ABB RAPID module: P50.mod

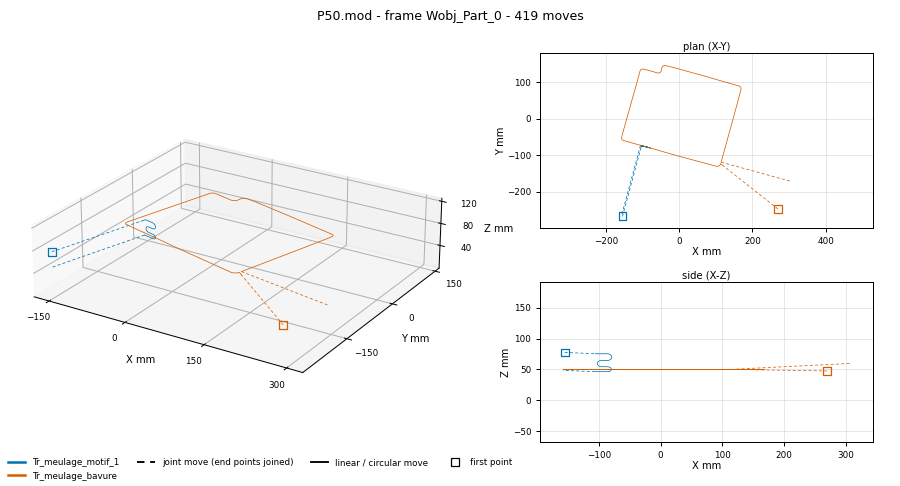
[picture p0: tool path of P50.mod in frame Wobj_Part_0, 419 of 426 moves have a stored position in this frame; points joined in program order, loops and branches not executed]
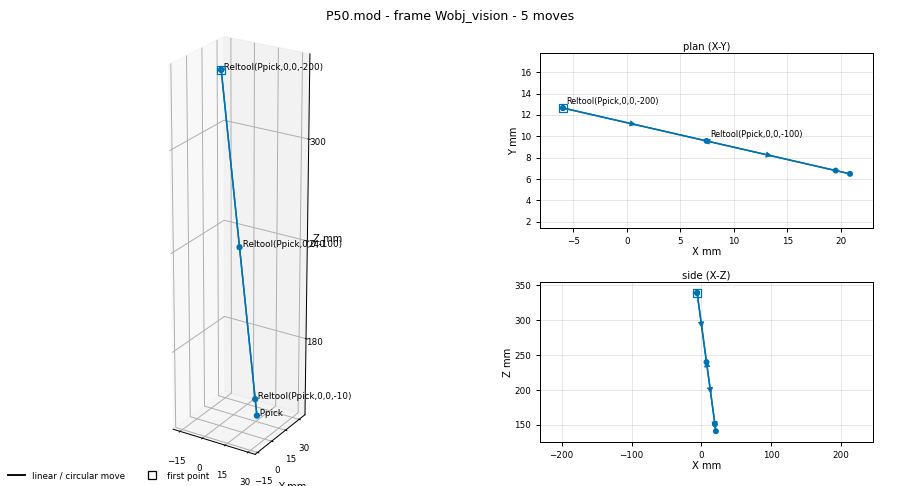
[picture p1: tool path of P50.mod in frame Wobj_vision, 5 of 426 moves have a stored position in this frame; points joined in program order, loops and branches not executed]
MODULE P50
	LOCAL CONST Speeddata vitesse_Tronconnage :=[10, 500, 0, 0];
	LOCAL CONST Robtarget Tr_meulage_motif_1_App1 :=[[-155.319755166464,-266.991909099729,77.372571942786],[0.697372246118371,-0.704623915003405,0.0931525017095072,-0.0921938185257175],[0,0,0,0],[8.999999E+09,8.999999E+09,8.999999E+09,8.999999E+09,8.999999E+09,8.999999E+09]];
	LOCAL CONST Robtarget Tr_meulage_motif_1_App2 :=[[-105.948658461448,-83.5290196737364,75.4071168783893],[0.697372246118371,-0.704623915003405,0.0931525017095072,-0.0921938185257175],[0,0,0,0],[8.999999E+09,8.999999E+09,8.999999E+09,8.999999E+09,8.999999E+09,8.999999E+09]];
	LOCAL CONST Robtarget Tr_meulage_motif_1_P0 :=[[-103.3501796875,-73.873078125,75.303671875],[0.697372246118371,-0.704623915003405,0.0931525017095072,-0.0921938185257175],[0,0,0,0],[8.999999E+09,8.999999E+09,8.999999E+09,8.999999E+09,8.999999E+09,8.999999E+09]];
	LOCAL CONST Robtarget Tr_meulage_motif_1_P1 :=[[-102.3816328125,-74.12190625,75.303671875],[0.697372246118371,-0.704623915003405,0.0931525017095072,-0.0921938185257175],[0,0,0,0],[8.999999E+09,8.999999E+09,8.999999E+09,8.999999E+09,8.999999E+09,8.999999E+09]];
	LOCAL CONST Robtarget Tr_meulage_motif_1_P2 :=[[-101.4130859375,-74.3707421875,75.303671875],[0.697372246118371,-0.704623915003405,0.0931525017095072,-0.0921938185257175],[0,0,0,0],[8.999999E+09,8.999999E+09,8.999999E+09,8.999999E+09,8.999999E+09,8.999999E+09]];
	LOCAL CONST Robtarget Tr_meulage_motif_1_P3 :=[[-100.4445390625,-74.6195703125,75.303671875],[0.697372246118371,-0.704623915003405,0.0931525017095072,-0.0921938185257175],[0,0,0,0],[8.999999E+09,8.999999E+09,8.999999E+09,8.999999E+09,8.999999E+09,8.999999E+09]];
	LOCAL CONST Robtarget Tr_meulage_motif_1_P4 :=[[-99.4759921875,-74.8683984375,75.303671875],[0.697372246118371,-0.704623915003405,0.0931525017095072,-0.0921938185257175],[0,0,0,0],[8.999999E+09,8.999999E+09,8.999999E+09,8.999999E+09,8.999999E+09,8.999999E+09]];
	LOCAL CONST Robtarget Tr_meulage_motif_1_P5 :=[[-98.5074453125,-75.117234375,75.303671875],[0.697372246118371,-0.704623915003405,0.0931525017095072,-0.0921938185257175],[0,0,0,0],[8.999999E+09,8.999999E+09,8.999999E+09,8.999999E+09,8.999999E+09,8.999999E+09]];
	LOCAL CONST Robtarget Tr_meulage_motif_1_P6 :=[[-97.5388984375,-75.3660625,75.303671875],[0.697372246118371,-0.704623915003405,0.0931525017095072,-0.0921938185257175],[0,0,0,0],[8.999999E+09,8.999999E+09,8.999999E+09,8.999999E+09,8.999999E+09,8.999999E+09]];
	LOCAL CONST Robtarget Tr_meulage_motif_1_P7 :=[[-96.5703515625,-75.6148984375,75.303671875],[0.697372246118371,-0.704623915003405,0.0931525017095072,-0.0921938185257175],[0,0,0,0],[8.999999E+09,8.999999E+09,8.999999E+09,8.999999E+09,8.999999E+09,8.999999E+09]];
	LOCAL CONST Robtarget Tr_meulage_motif_1_P8 :=[[-95.6018046875,-75.8637265625,75.303671875],[0.697372246118371,-0.704623915003405,0.0931525017095072,-0.0921938185257175],[0,0,0,0],[8.999999E+09,8.999999E+09,8.999999E+09,8.999999E+09,8.999999E+09,8.999999E+09]];
	LOCAL CONST Robtarget Tr_meulage_motif_1_P9 :=[[-94.6332578125,-76.1125546875,75.3036796875],[0.697372246118371,-0.704623915003405,0.0931525017095072,-0.0921938185257175],[0,0,0,0],[8.999999E+09,8.999999E+09,8.999999E+09,8.999999E+09,8.999999E+09,8.999999E+09]];
	LOCAL CONST Robtarget Tr_meulage_motif_1_P10 :=[[-93.6647109375,-76.361390625,75.3036796875],[0.697372246118371,-0.704623915003405,0.0931525017095072,-0.0921938185257175],[0,0,0,0],[8.999999E+09,8.999999E+09,8.999999E+09,8.999999E+09,8.999999E+09,8.999999E+09]];
	LOCAL CONST Robtarget Tr_meulage_motif_1_P11 :=[[-92.6961640625,-76.61021875,75.3036796875],[0.697372246118371,-0.704623915003405,0.0931525017095072,-0.0921938185257175],[0,0,0,0],[8.999999E+09,8.999999E+09,8.999999E+09,8.999999E+09,8.999999E+09,8.999999E+09]];
	LOCAL CONST Robtarget Tr_meulage_motif_1_P12 :=[[-91.7276171875,-76.8590546875,75.3036796875],[0.697372246118371,-0.704623915003405,0.0931525017095072,-0.0921938185257175],[0,0,0,0],[8.999999E+09,8.999999E+09,8.999999E+09,8.999999E+09,8.999999E+09,8.999999E+09]];
	LOCAL CONST Robtarget Tr_meulage_motif_1_P13 :=[[-90.7590703125,-77.1078828125,75.3036796875],[0.697372246118371,-0.704623915003405,0.0931525017095072,-0.0921938185257175],[0,0,0,0],[8.999999E+09,8.999999E+09,8.999999E+09,8.999999E+09,8.999999E+09,8.999999E+09]];
	LOCAL CONST Robtarget Tr_meulage_motif_1_P14 :=[[-89.7905234375,-77.3567109375,75.3036796875],[0.697372246118371,-0.704623915003405,0.0931525017095072,-0.0921938185257175],[0,0,0,0],[8.999999E+09,8.999999E+09,8.999999E+09,8.999999E+09,8.999999E+09,8.999999E+09]];
	LOCAL CONST Robtarget Tr_meulage_motif_1_P15 :=[[-88.8219765625,-77.605546875,75.3036796875],[0.697372246118371,-0.704623915003405,0.0931525017095072,-0.0921938185257175],[0,0,0,0],[8.999999E+09,8.999999E+09,8.999999E+09,8.999999E+09,8.999999E+09,8.999999E+09]];
	LOCAL CONST Robtarget Tr_meulage_motif_1_P16 :=[[-87.8534296875,-77.854375,75.3036796875],[0.697372246118371,-0.704623915003405,0.0931525017095072,-0.0921938185257175],[0,0,0,0],[8.999999E+09,8.999999E+09,8.999999E+09,8.999999E+09,8.999999E+09,8.999999E+09]];
	LOCAL CONST Robtarget Tr_meulage_motif_1_P17 :=[[-86.8848828125,-78.1032109375,75.3036796875],[0.697372246118371,-0.704623915003405,0.0931525017095072,-0.0921938185257175],[0,0,0,0],[8.999999E+09,8.999999E+09,8.999999E+09,8.999999E+09,8.999999E+09,8.999999E+09]];
	LOCAL CONST Robtarget Tr_meulage_motif_1_P18 :=[[-85.9163359375,-78.3520390625,75.3036796875],[0.697372246118371,-0.704623915003405,0.0931525017095072,-0.0921938185257175],[0,0,0,0],[8.999999E+09,8.999999E+09,8.999999E+09,8.999999E+09,8.999999E+09,8.999999E+09]];
	LOCAL CONST Robtarget Tr_meulage_motif_1_P19 :=[[-84.95490625,-78.5986953125,75.1930859375],[0.697372246118371,-0.704623915003405,0.0931525017095072,-0.0921938185257175],[0,0,0,0],[8.999999E+09,8.999999E+09,8.999999E+09,8.999999E+09,8.999999E+09,8.999999E+09]];
	LOCAL CONST Robtarget Tr_meulage_motif_1_P20 :=[[-84.0380234375,-78.83359375,74.9818984375],[0.697372246118371,-0.704623915003405,0.0931525017095072,-0.0921938185257175],[0,0,0,0],[8.999999E+09,8.999999E+09,8.999999E+09,8.999999E+09,8.999999E+09,8.999999E+09]];
	LOCAL CONST Robtarget Tr_meulage_motif_1_P21 :=[[-83.211921875,-79.044984375,74.7100546875],[0.697372246118371,-0.704623915003405,0.0931525017095072,-0.0921938185257175],[0,0,0,0],[8.999999E+09,8.999999E+09,8.999999E+09,8.999999E+09,8.999999E+09,8.999999E+09]];
	LOCAL CONST Robtarget Tr_meulage_motif_1_P22 :=[[-82.485359375,-79.23078125,74.4341171875],[0.697372246118371,-0.704623915003405,0.0931525017095072,-0.0921938185257175],[0,0,0,0],[8.999999E+09,8.999999E+09,8.999999E+09,8.999999E+09,8.999999E+09,8.999999E+09]];
	LOCAL CONST Robtarget Tr_meulage_motif_1_P23 :=[[-81.41846875,-79.5029609375,73.8179921875],[0.697372246118371,-0.704623915003405,0.0931525017095072,-0.0921938185257175],[0,0,0,0],[8.999999E+09,8.999999E+09,8.999999E+09,8.999999E+09,8.999999E+09,8.999999E+09]];
	LOCAL CONST Robtarget Tr_meulage_motif_1_P24 :=[[-80.42615625,-79.75525,72.97034375],[0.697372246118371,-0.704623915003405,0.0931525017095072,-0.0921938185257175],[0,0,0,0],[8.999999E+09,8.999999E+09,8.999999E+09,8.999999E+09,8.999999E+09,8.999999E+09]];
	LOCAL CONST Robtarget Tr_meulage_motif_1_P25 :=[[-79.604390625,-79.963171875,71.9464765625],[0.697372246118371,-0.704623915003405,0.0931525017095072,-0.0921938185257175],[0,0,0,0],[8.999999E+09,8.999999E+09,8.999999E+09,8.999999E+09,8.999999E+09,8.999999E+09]];
	LOCAL CONST Robtarget Tr_meulage_motif_1_P26 :=[[-79.13075,-80.081375,70.8302890625],[0.697372246118371,-0.704623915003405,0.0931525017095072,-0.0921938185257175],[0,0,0,0],[8.999999E+09,8.999999E+09,8.999999E+09,8.999999E+09,8.999999E+09,8.999999E+09]];
	LOCAL CONST Robtarget Tr_meulage_motif_1_P27 :=[[-79.104015625,-80.0860703125,70.134328125],[0.697372246118371,-0.704623915003405,0.0931525017095072,-0.0921938185257175],[0,0,0,0],[8.999999E+09,8.999999E+09,8.999999E+09,8.999999E+09,8.999999E+09,8.999999E+09]];
	LOCAL CONST Robtarget Tr_meulage_motif_1_P28 :=[[-79.103515625,-80.0841328125,69.473078125],[0.697372246118371,-0.704623915003405,0.0931525017095072,-0.0921938185257175],[0,0,0,0],[8.999999E+09,8.999999E+09,8.999999E+09,8.999999E+09,8.999999E+09,8.999999E+09]];
	LOCAL CONST Robtarget Tr_meulage_motif_1_P29 :=[[-79.156171875,-80.0685390625,68.811984375],[0.697372246118371,-0.704623915003405,0.0931525017095072,-0.0921938185257175],[0,0,0,0],[8.999999E+09,8.999999E+09,8.999999E+09,8.999999E+09,8.999999E+09,8.999999E+09]];
	LOCAL CONST Robtarget Tr_meulage_motif_1_P30 :=[[-79.637890625,-79.94134375,67.7102421875],[0.697372246118371,-0.704623915003405,0.0931525017095072,-0.0921938185257175],[0,0,0,0],[8.999999E+09,8.999999E+09,8.999999E+09,8.999999E+09,8.999999E+09,8.999999E+09]];
	LOCAL CONST Robtarget Tr_meulage_motif_1_P31 :=[[-80.4668125,-79.7252421875,66.703625],[0.697372246118371,-0.704623915003405,0.0931525017095072,-0.0921938185257175],[0,0,0,0],[8.999999E+09,8.999999E+09,8.999999E+09,8.999999E+09,8.999999E+09,8.999999E+09]];
	LOCAL CONST Robtarget Tr_meulage_motif_1_P32 :=[[-81.45740625,-79.46815625,65.87475],[0.697372246118371,-0.704623915003405,0.0931525017095072,-0.0921938185257175],[0,0,0,0],[8.999999E+09,8.999999E+09,8.999999E+09,8.999999E+09,8.999999E+09,8.999999E+09]];
	LOCAL CONST Robtarget Tr_meulage_motif_1_P33 :=[[-82.12259375,-79.29603125,65.47900390625],[0.697372246118371,-0.704623915003405,0.0931525017095072,-0.0921938185257175],[0,0,0,0],[8.999999E+09,8.999999E+09,8.999999E+09,8.999999E+09,8.999999E+09,8.999999E+09]];
	LOCAL CONST Robtarget Tr_meulage_motif_1_P34 :=[[-83.243953125,-79.0064140625,64.99147265625],[0.697372246118371,-0.704623915003405,0.0931525017095072,-0.0921938185257175],[0,0,0,0],[8.999999E+09,8.999999E+09,8.999999E+09,8.999999E+09,8.999999E+09,8.999999E+09]];
	LOCAL CONST Robtarget Tr_meulage_motif_1_P35 :=[[-84.0622109375,-78.795375,64.7273828125],[0.697372246118371,-0.704623915003405,0.0931525017095072,-0.0921938185257175],[0,0,0,0],[8.999999E+09,8.999999E+09,8.999999E+09,8.999999E+09,8.999999E+09,8.999999E+09]];
	LOCAL CONST Robtarget Tr_meulage_motif_1_P36 :=[[-84.9647421875,-78.562859375,64.5229140625],[0.697372246118371,-0.704623915003405,0.0931525017095072,-0.0921938185257175],[0,0,0,0],[8.999999E+09,8.999999E+09,8.999999E+09,8.999999E+09,8.999999E+09,8.999999E+09]];
	LOCAL CONST Robtarget Tr_meulage_motif_1_P37 :=[[-85.91534375,-78.318296875,64.4143203125],[0.697372246118371,-0.704623915003405,0.0931525017095072,-0.0921938185257175],[0,0,0,0],[8.999999E+09,8.999999E+09,8.999999E+09,8.999999E+09,8.999999E+09,8.999999E+09]];
	LOCAL CONST Robtarget Tr_meulage_motif_1_P38 :=[[-86.876609375,-78.0709921875,64.3037265625],[0.697372246118371,-0.704623915003405,0.0931525017095072,-0.0921938185257175],[0,0,0,0],[8.999999E+09,8.999999E+09,8.999999E+09,8.999999E+09,8.999999E+09,8.999999E+09]];
	LOCAL CONST Robtarget Tr_meulage_motif_1_P39 :=[[-87.84515625,-77.8221640625,64.3037265625],[0.697372246118371,-0.704623915003405,0.0931525017095072,-0.0921938185257175],[0,0,0,0],[8.999999E+09,8.999999E+09,8.999999E+09,8.999999E+09,8.999999E+09,8.999999E+09]];
	LOCAL CONST Robtarget Tr_meulage_motif_1_P40 :=[[-88.813703125,-77.5733359375,64.3037265625],[0.697372246118371,-0.704623915003405,0.0931525017095072,-0.0921938185257175],[0,0,0,0],[8.999999E+09,8.999999E+09,8.999999E+09,8.999999E+09,8.999999E+09,8.999999E+09]];
	LOCAL CONST Robtarget Tr_meulage_motif_1_P41 :=[[-89.78225,-77.3245,64.3037265625],[0.697372246118371,-0.704623915003405,0.0931525017095072,-0.0921938185257175],[0,0,0,0],[8.999999E+09,8.999999E+09,8.999999E+09,8.999999E+09,8.999999E+09,8.999999E+09]];
	LOCAL CONST Robtarget Tr_meulage_motif_1_P42 :=[[-90.750796875,-77.075671875,64.3037265625],[0.697372246118371,-0.704623915003405,0.0931525017095072,-0.0921938185257175],[0,0,0,0],[8.999999E+09,8.999999E+09,8.999999E+09,8.999999E+09,8.999999E+09,8.999999E+09]];
	LOCAL CONST Robtarget Tr_meulage_motif_1_P43 :=[[-91.71934375,-76.82684375,64.3037265625],[0.697372246118371,-0.704623915003405,0.0931525017095072,-0.0921938185257175],[0,0,0,0],[8.999999E+09,8.999999E+09,8.999999E+09,8.999999E+09,8.999999E+09,8.999999E+09]];
	LOCAL CONST Robtarget Tr_meulage_motif_1_P44 :=[[-92.687890625,-76.5780078125,64.3037265625],[0.697372246118371,-0.704623915003405,0.0931525017095072,-0.0921938185257175],[0,0,0,0],[8.999999E+09,8.999999E+09,8.999999E+09,8.999999E+09,8.999999E+09,8.999999E+09]];
	LOCAL CONST Robtarget Tr_meulage_motif_1_P45 :=[[-93.6564375,-76.3291796875,64.3037265625],[0.697372246118371,-0.704623915003405,0.0931525017095072,-0.0921938185257175],[0,0,0,0],[8.999999E+09,8.999999E+09,8.999999E+09,8.999999E+09,8.999999E+09,8.999999E+09]];
	LOCAL CONST Robtarget Tr_meulage_motif_1_P46 :=[[-94.624984375,-76.08034375,64.3037265625],[0.697372246118371,-0.704623915003405,0.0931525017095072,-0.0921938185257175],[0,0,0,0],[8.999999E+09,8.999999E+09,8.999999E+09,8.999999E+09,8.999999E+09,8.999999E+09]];
	LOCAL CONST Robtarget Tr_meulage_motif_1_P47 :=[[-95.59353125,-75.831515625,64.3037265625],[0.697372246118371,-0.704623915003405,0.0931525017095072,-0.0921938185257175],[0,0,0,0],[8.999999E+09,8.999999E+09,8.999999E+09,8.999999E+09,8.999999E+09,8.999999E+09]];
	LOCAL CONST Robtarget Tr_meulage_motif_1_P48 :=[[-96.562078125,-75.5826875,64.3037265625],[0.697372246118371,-0.704623915003405,0.0931525017095072,-0.0921938185257175],[0,0,0,0],[8.999999E+09,8.999999E+09,8.999999E+09,8.999999E+09,8.999999E+09,8.999999E+09]];
	LOCAL CONST Robtarget Tr_meulage_motif_1_P49 :=[[-97.5233359375,-75.3353828125,64.1931328125],[0.697372246118371,-0.704623915003405,0.0931525017095072,-0.0921938185257175],[0,0,0,0],[8.999999E+09,8.999999E+09,8.999999E+09,8.999999E+09,8.999999E+09,8.999999E+09]];
	LOCAL CONST Robtarget Tr_meulage_motif_1_P50 :=[[-98.43990625,-75.0992421875,63.9819453125],[0.697372246118371,-0.704623915003405,0.0931525017095072,-0.0921938185257175],[0,0,0,0],[8.999999E+09,8.999999E+09,8.999999E+09,8.999999E+09,8.999999E+09,8.999999E+09]];
	LOCAL CONST Robtarget Tr_meulage_motif_1_P51 :=[[-99.2656015625,-74.886265625,63.71010546875],[0.697372246118371,-0.704623915003405,0.0931525017095072,-0.0921938185257175],[0,0,0,0],[8.999999E+09,8.999999E+09,8.999999E+09,8.999999E+09,8.999999E+09,8.999999E+09]];
	LOCAL CONST Robtarget Tr_meulage_motif_1_P52 :=[[-99.9544921875,-74.708328125,63.40594921875],[0.697372246118371,-0.704623915003405,0.0931525017095072,-0.0921938185257175],[0,0,0,0],[8.999999E+09,8.999999E+09,8.999999E+09,8.999999E+09,8.999999E+09,8.999999E+09]];
	LOCAL CONST Robtarget Tr_meulage_motif_1_P53 :=[[-100.955921875,-74.448984375,62.743421875],[0.697372246118371,-0.704623915003405,0.0931525017095072,-0.0921938185257175],[0,0,0,0],[8.999999E+09,8.999999E+09,8.999999E+09,8.999999E+09,8.999999E+09,8.999999E+09]];
	LOCAL CONST Robtarget Tr_meulage_motif_1_P54 :=[[-101.8288125,-74.22190625,61.84148828125],[0.697372246118371,-0.704623915003405,0.0931525017095072,-0.0921938185257175],[0,0,0,0],[8.999999E+09,8.999999E+09,8.999999E+09,8.999999E+09,8.999999E+09,8.999999E+09]];
	LOCAL CONST Robtarget Tr_meulage_motif_1_P55 :=[[-102.346171875,-74.0857265625,60.7954609375],[0.697372246118371,-0.704623915003405,0.0931525017095072,-0.0921938185257175],[0,0,0,0],[8.999999E+09,8.999999E+09,8.999999E+09,8.999999E+09,8.999999E+09,8.999999E+09]];
	LOCAL CONST Robtarget Tr_meulage_motif_1_P56 :=[[-102.5246171875,-74.03771875,60.10224609375],[0.697372246118371,-0.704623915003405,0.0931525017095072,-0.0921938185257175],[0,0,0,0],[8.999999E+09,8.999999E+09,8.999999E+09,8.999999E+09,8.999999E+09,8.999999E+09]];
	LOCAL CONST Robtarget Tr_meulage_motif_1_P57 :=[[-102.585875,-74.019578125,59.33225],[0.697372246118371,-0.704623915003405,0.0931525017095072,-0.0921938185257175],[0,0,0,0],[8.999999E+09,8.999999E+09,8.999999E+09,8.999999E+09,8.999999E+09,8.999999E+09]];
	LOCAL CONST Robtarget Tr_meulage_motif_1_P58 :=[[-102.5204609375,-74.033984375,58.562375],[0.697372246118371,-0.704623915003405,0.0931525017095072,-0.0921938185257175],[0,0,0,0],[8.999999E+09,8.999999E+09,8.999999E+09,8.999999E+09,8.999999E+09,8.999999E+09]];
	LOCAL CONST Robtarget Tr_meulage_motif_1_P59 :=[[-102.113234375,-74.135140625,57.4541328125],[0.697372246118371,-0.704623915003405,0.0931525017095072,-0.0921938185257175],[0,0,0,0],[8.999999E+09,8.999999E+09,8.999999E+09,8.999999E+09,8.999999E+09,8.999999E+09]];
	LOCAL CONST Robtarget Tr_meulage_motif_1_P60 :=[[-101.7115078125,-74.2365234375,56.8684453125],[0.697372246118371,-0.704623915003405,0.0931525017095072,-0.0921938185257175],[0,0,0,0],[8.999999E+09,8.999999E+09,8.999999E+09,8.999999E+09,8.999999E+09,8.999999E+09]];
	LOCAL CONST Robtarget Tr_meulage_motif_1_P61 :=[[-100.851625,-74.454671875,55.981328125],[0.697372246118371,-0.704623915003405,0.0931525017095072,-0.0921938185257175],[0,0,0,0],[8.999999E+09,8.999999E+09,8.999999E+09,8.999999E+09,8.999999E+09,8.999999E+09]];
	LOCAL CONST Robtarget Tr_meulage_motif_1_P62 :=[[-100.284046875,-74.5991953125,55.567015625],[0.697372246118371,-0.704623915003405,0.0931525017095072,-0.0921938185257175],[0,0,0,0],[8.999999E+09,8.999999E+09,8.999999E+09,8.999999E+09,8.999999E+09,8.999999E+09]];
	LOCAL CONST Robtarget Tr_meulage_motif_1_P63 :=[[-99.200890625,-74.875765625,55.02292578125],[0.697372246118371,-0.704623915003405,0.0931525017095072,-0.0921938185257175],[0,0,0,0],[8.999999E+09,8.999999E+09,8.999999E+09,8.999999E+09,8.999999E+09,8.999999E+09]];
	LOCAL CONST Robtarget Tr_meulage_motif_1_P64 :=[[-98.4010390625,-75.0803359375,54.72742578125],[0.697372246118371,-0.704623915003405,0.0931525017095072,-0.0921938185257175],[0,0,0,0],[8.999999E+09,8.999999E+09,8.999999E+09,8.999999E+09,8.999999E+09,8.999999E+09]];
	LOCAL CONST Robtarget Tr_meulage_motif_1_P65 :=[[-97.498203125,-75.3116484375,54.52295703125],[0.697372246118371,-0.704623915003405,0.0931525017095072,-0.0921938185257175],[0,0,0,0],[8.999999E+09,8.999999E+09,8.999999E+09,8.999999E+09,8.999999E+09,8.999999E+09]];
	LOCAL CONST Robtarget Tr_meulage_motif_1_P66 :=[[-96.5474296875,-75.555578125,54.41436328125],[0.697372246118371,-0.704623915003405,0.0931525017095072,-0.0921938185257175],[0,0,0,0],[8.999999E+09,8.999999E+09,8.999999E+09,8.999999E+09,8.999999E+09,8.999999E+09]];
	LOCAL CONST Robtarget Tr_meulage_motif_1_P67 :=[[-95.5860078125,-75.802234375,54.3037734375],[0.697372246118371,-0.704623915003405,0.0931525017095072,-0.0921938185257175],[0,0,0,0],[8.999999E+09,8.999999E+09,8.999999E+09,8.999999E+09,8.999999E+09,8.999999E+09]];
	LOCAL CONST Robtarget Tr_meulage_motif_1_P68 :=[[-94.6174609375,-76.0510625,54.3037734375],[0.697372246118371,-0.704623915003405,0.0931525017095072,-0.0921938185257175],[0,0,0,0],[8.999999E+09,8.999999E+09,8.999999E+09,8.999999E+09,8.999999E+09,8.999999E+09]];
	LOCAL CONST Robtarget Tr_meulage_motif_1_P69 :=[[-93.6489140625,-76.299890625,54.3037734375],[0.697372246118371,-0.704623915003405,0.0931525017095072,-0.0921938185257175],[0,0,0,0],[8.999999E+09,8.999999E+09,8.999999E+09,8.999999E+09,8.999999E+09,8.999999E+09]];
	LOCAL CONST Robtarget Tr_meulage_motif_1_P70 :=[[-92.6803671875,-76.5487265625,54.3037734375],[0.697372246118371,-0.704623915003405,0.0931525017095072,-0.0921938185257175],[0,0,0,0],[8.999999E+09,8.999999E+09,8.999999E+09,8.999999E+09,8.999999E+09,8.999999E+09]];
	LOCAL CONST Robtarget Tr_meulage_motif_1_P71 :=[[-91.7118203125,-76.7975546875,54.3037734375],[0.697372246118371,-0.704623915003405,0.0931525017095072,-0.0921938185257175],[0,0,0,0],[8.999999E+09,8.999999E+09,8.999999E+09,8.999999E+09,8.999999E+09,8.999999E+09]];
	LOCAL CONST Robtarget Tr_meulage_motif_1_P72 :=[[-90.7432734375,-77.046390625,54.3037734375],[0.697372246118371,-0.704623915003405,0.0931525017095072,-0.0921938185257175],[0,0,0,0],[8.999999E+09,8.999999E+09,8.999999E+09,8.999999E+09,8.999999E+09,8.999999E+09]];
	LOCAL CONST Robtarget Tr_meulage_motif_1_P73 :=[[-89.7747265625,-77.29521875,54.3037734375],[0.697372246118371,-0.704623915003405,0.0931525017095072,-0.0921938185257175],[0,0,0,0],[8.999999E+09,8.999999E+09,8.999999E+09,8.999999E+09,8.999999E+09,8.999999E+09]];
	LOCAL CONST Robtarget Tr_meulage_motif_1_P74 :=[[-88.8061796875,-77.544046875,54.3037734375],[0.697372246118371,-0.704623915003405,0.0931525017095072,-0.0921938185257175],[0,0,0,0],[8.999999E+09,8.999999E+09,8.999999E+09,8.999999E+09,8.999999E+09,8.999999E+09]];
	LOCAL CONST Robtarget Tr_meulage_motif_1_P75 :=[[-87.8376328125,-77.7928828125,54.3037734375],[0.697372246118371,-0.704623915003405,0.0931525017095072,-0.0921938185257175],[0,0,0,0],[8.999999E+09,8.999999E+09,8.999999E+09,8.999999E+09,8.999999E+09,8.999999E+09]];
	LOCAL CONST Robtarget Tr_meulage_motif_1_P76 :=[[-86.8690859375,-78.0417109375,54.3037734375],[0.697372246118371,-0.704623915003405,0.0931525017095072,-0.0921938185257175],[0,0,0,0],[8.999999E+09,8.999999E+09,8.999999E+09,8.999999E+09,8.999999E+09,8.999999E+09]];
	LOCAL CONST Robtarget Tr_meulage_motif_1_P77 :=[[-85.9005390625,-78.290546875,54.3037734375],[0.697372246118371,-0.704623915003405,0.0931525017095072,-0.0921938185257175],[0,0,0,0],[8.999999E+09,8.999999E+09,8.999999E+09,8.999999E+09,8.999999E+09,8.999999E+09]];
	LOCAL CONST Robtarget Tr_meulage_motif_1_P78 :=[[-84.939109375,-78.537203125,54.1931796875],[0.697372246118371,-0.704623915003405,0.0931525017095072,-0.0921938185257175],[0,0,0,0],[8.999999E+09,8.999999E+09,8.999999E+09,8.999999E+09,8.999999E+09,8.999999E+09]];
	LOCAL CONST Robtarget Tr_meulage_motif_1_P79 :=[[-84.02221875,-78.7721015625,53.9819921875],[0.697372246118371,-0.704623915003405,0.0931525017095072,-0.0921938185257175],[0,0,0,0],[8.999999E+09,8.999999E+09,8.999999E+09,8.999999E+09,8.999999E+09,8.999999E+09]];
	LOCAL CONST Robtarget Tr_meulage_motif_1_P80 :=[[-83.1961171875,-78.983484375,53.7101484375],[0.697372246118371,-0.704623915003405,0.0931525017095072,-0.0921938185257175],[0,0,0,0],[8.999999E+09,8.999999E+09,8.999999E+09,8.999999E+09,8.999999E+09,8.999999E+09]];
	LOCAL CONST Robtarget Tr_meulage_motif_1_P81 :=[[-82.4695625,-79.1692890625,53.43421484375],[0.697372246118371,-0.704623915003405,0.0931525017095072,-0.0921938185257175],[0,0,0,0],[8.999999E+09,8.999999E+09,8.999999E+09,8.999999E+09,8.999999E+09,8.999999E+09]];
	LOCAL CONST Robtarget Tr_meulage_motif_1_P82 :=[[-81.4026640625,-79.4414609375,52.81809375],[0.697372246118371,-0.704623915003405,0.0931525017095072,-0.0921938185257175],[0,0,0,0],[8.999999E+09,8.999999E+09,8.999999E+09,8.999999E+09,8.999999E+09,8.999999E+09]];
	LOCAL CONST Robtarget Tr_meulage_motif_1_P83 :=[[-80.4753671875,-79.67690625,51.92412890625],[0.697372246118371,-0.704623915003405,0.0931525017095072,-0.0921938185257175],[0,0,0,0],[8.999999E+09,8.999999E+09,8.999999E+09,8.999999E+09,8.999999E+09,8.999999E+09]];
	LOCAL CONST Robtarget Tr_meulage_motif_1_P84 :=[[-79.8845859375,-79.825296875,50.8381328125],[0.697372246118371,-0.704623915003405,0.0931525017095072,-0.0921938185257175],[0,0,0,0],[8.999999E+09,8.999999E+09,8.999999E+09,8.999999E+09,8.999999E+09,8.999999E+09]];
	LOCAL CONST Robtarget Tr_meulage_motif_1_P85 :=[[-79.719859375,-79.8645390625,49.85376171875],[0.697372246118371,-0.704623915003405,0.0931525017095072,-0.0921938185257175],[0,0,0,0],[8.999999E+09,8.999999E+09,8.999999E+09,8.999999E+09,8.999999E+09,8.999999E+09]];
	LOCAL CONST Robtarget Tr_meulage_motif_1_P86 :=[[-79.8470390625,-79.8312265625,49.64910546875],[0.697372246118371,-0.704623915003405,0.0931525017095072,-0.0921938185257175],[0,0,0,0],[8.999999E+09,8.999999E+09,8.999999E+09,8.999999E+09,8.999999E+09,8.999999E+09]];
	LOCAL CONST Robtarget Tr_meulage_motif_1_P87 :=[[-79.965984375,-79.79840625,48.922703125],[0.697372246118371,-0.704623915003405,0.0931525017095072,-0.0921938185257175],[0,0,0,0],[8.999999E+09,8.999999E+09,8.999999E+09,8.999999E+09,8.999999E+09,8.999999E+09]];
	LOCAL CONST Robtarget Tr_meulage_motif_1_P88 :=[[-80.627765625,-79.6254609375,47.98580078125],[0.697372246118371,-0.704623915003405,0.0931525017095072,-0.0921938185257175],[0,0,0,0],[8.999999E+09,8.999999E+09,8.999999E+09,8.999999E+09,8.999999E+09,8.999999E+09]];
	LOCAL CONST Robtarget Tr_meulage_motif_1_P89 :=[[-81.1675,-79.48534375,47.5219921875],[0.697372246118371,-0.704623915003405,0.0931525017095072,-0.0921938185257175],[0,0,0,0],[8.999999E+09,8.999999E+09,8.999999E+09,8.999999E+09,8.999999E+09,8.999999E+09]];
	LOCAL CONST Robtarget Tr_meulage_motif_1_P90 :=[[-82.2618671875,-79.2025390625,46.9915546875],[0.697372246118371,-0.704623915003405,0.0931525017095072,-0.0921938185257175],[0,0,0,0],[8.999999E+09,8.999999E+09,8.999999E+09,8.999999E+09,8.999999E+09,8.999999E+09]];
	LOCAL CONST Robtarget Tr_meulage_motif_1_P91 :=[[-83.0801171875,-78.9914921875,46.72746484375],[0.697372246118371,-0.704623915003405,0.0931525017095072,-0.0921938185257175],[0,0,0,0],[8.999999E+09,8.999999E+09,8.999999E+09,8.999999E+09,8.999999E+09,8.999999E+09]];
	LOCAL CONST Robtarget Tr_meulage_motif_1_P92 :=[[-83.9826484375,-78.758984375,46.52299609375],[0.697372246118371,-0.704623915003405,0.0931525017095072,-0.0921938185257175],[0,0,0,0],[8.999999E+09,8.999999E+09,8.999999E+09,8.999999E+09,8.999999E+09,8.999999E+09]];
	LOCAL CONST Robtarget Tr_meulage_motif_1_P93 :=[[-84.9332578125,-78.514421875,46.41440234375],[0.697372246118371,-0.704623915003405,0.0931525017095072,-0.0921938185257175],[0,0,0,0],[8.999999E+09,8.999999E+09,8.999999E+09,8.999999E+09,8.999999E+09,8.999999E+09]];
	LOCAL CONST Robtarget Tr_meulage_motif_1_P94 :=[[-85.894515625,-78.2671171875,46.30380859375],[0.697372246118371,-0.704623915003405,0.0931525017095072,-0.0921938185257175],[0,0,0,0],[8.999999E+09,8.999999E+09,8.999999E+09,8.999999E+09,8.999999E+09,8.999999E+09]];
	LOCAL CONST Robtarget Tr_meulage_motif_1_P95 :=[[-86.8630625,-78.0182890625,46.30380859375],[0.697372246118371,-0.704623915003405,0.0931525017095072,-0.0921938185257175],[0,0,0,0],[8.999999E+09,8.999999E+09,8.999999E+09,8.999999E+09,8.999999E+09,8.999999E+09]];
	LOCAL CONST Robtarget Tr_meulage_motif_1_P96 :=[[-87.831609375,-77.769453125,46.30380859375],[0.697372246118371,-0.704623915003405,0.0931525017095072,-0.0921938185257175],[0,0,0,0],[8.999999E+09,8.999999E+09,8.999999E+09,8.999999E+09,8.999999E+09,8.999999E+09]];
	LOCAL CONST Robtarget Tr_meulage_motif_1_P97 :=[[-88.80015625,-77.520625,46.30380859375],[0.697372246118371,-0.704623915003405,0.0931525017095072,-0.0921938185257175],[0,0,0,0],[8.999999E+09,8.999999E+09,8.999999E+09,8.999999E+09,8.999999E+09,8.999999E+09]];
	LOCAL CONST Robtarget Tr_meulage_motif_1_P98 :=[[-89.768703125,-77.2717890625,46.30380859375],[0.697372246118371,-0.704623915003405,0.0931525017095072,-0.0921938185257175],[0,0,0,0],[8.999999E+09,8.999999E+09,8.999999E+09,8.999999E+09,8.999999E+09,8.999999E+09]];
	LOCAL CONST Robtarget Tr_meulage_motif_1_P99 :=[[-90.73725,-77.0229609375,46.30380859375],[0.697372246118371,-0.704623915003405,0.0931525017095072,-0.0921938185257175],[0,0,0,0],[8.999999E+09,8.999999E+09,8.999999E+09,8.999999E+09,8.999999E+09,8.999999E+09]];
	LOCAL CONST Robtarget Tr_meulage_motif_1_P100 :=[[-91.705796875,-76.7741328125,46.30380859375],[0.697372246118371,-0.704623915003405,0.0931525017095072,-0.0921938185257175],[0,0,0,0],[8.999999E+09,8.999999E+09,8.999999E+09,8.999999E+09,8.999999E+09,8.999999E+09]];
	LOCAL CONST Robtarget Tr_meulage_motif_1_P101 :=[[-92.67434375,-76.525296875,46.30380859375],[0.697372246118371,-0.704623915003405,0.0931525017095072,-0.0921938185257175],[0,0,0,0],[8.999999E+09,8.999999E+09,8.999999E+09,8.999999E+09,8.999999E+09,8.999999E+09]];
	LOCAL CONST Robtarget Tr_meulage_motif_1_P102 :=[[-93.642890625,-76.27646875,46.30380859375],[0.697372246118371,-0.704623915003405,0.0931525017095072,-0.0921938185257175],[0,0,0,0],[8.999999E+09,8.999999E+09,8.999999E+09,8.999999E+09,8.999999E+09,8.999999E+09]];
	LOCAL CONST Robtarget Tr_meulage_motif_1_P103 :=[[-94.6114375,-76.0276328125,46.30380859375],[0.697372246118371,-0.704623915003405,0.0931525017095072,-0.0921938185257175],[0,0,0,0],[8.999999E+09,8.999999E+09,8.999999E+09,8.999999E+09,8.999999E+09,8.999999E+09]];
	LOCAL CONST Robtarget Tr_meulage_motif_1_P104 :=[[-95.579984375,-75.7788046875,46.30380859375],[0.697372246118371,-0.704623915003405,0.0931525017095072,-0.0921938185257175],[0,0,0,0],[8.999999E+09,8.999999E+09,8.999999E+09,8.999999E+09,8.999999E+09,8.999999E+09]];
	LOCAL CONST Robtarget Tr_meulage_motif_1_P105 :=[[-96.54853125,-75.5299765625,46.30380859375],[0.697372246118371,-0.704623915003405,0.0931525017095072,-0.0921938185257175],[0,0,0,0],[8.999999E+09,8.999999E+09,8.999999E+09,8.999999E+09,8.999999E+09,8.999999E+09]];
	LOCAL CONST Robtarget Tr_meulage_motif_1_P106 :=[[-97.517078125,-75.281140625,46.30380859375],[0.697372246118371,-0.704623915003405,0.0931525017095072,-0.0921938185257175],[0,0,0,0],[8.999999E+09,8.999999E+09,8.999999E+09,8.999999E+09,8.999999E+09,8.999999E+09]];
	LOCAL CONST Robtarget Tr_meulage_motif_1_P107 :=[[-98.485625,-75.0323125,46.30380859375],[0.697372246118371,-0.704623915003405,0.0931525017095072,-0.0921938185257175],[0,0,0,0],[8.999999E+09,8.999999E+09,8.999999E+09,8.999999E+09,8.999999E+09,8.999999E+09]];
	LOCAL CONST Robtarget Tr_meulage_motif_1_P108 :=[[-99.454171875,-74.7834765625,46.30380859375],[0.697372246118371,-0.704623915003405,0.0931525017095072,-0.0921938185257175],[0,0,0,0],[8.999999E+09,8.999999E+09,8.999999E+09,8.999999E+09,8.999999E+09,8.999999E+09]];
	LOCAL CONST Robtarget Tr_meulage_motif_1_P109 :=[[-100.42271875,-74.5346484375,46.30380859375],[0.697372246118371,-0.704623915003405,0.0931525017095072,-0.0921938185257175],[0,0,0,0],[8.999999E+09,8.999999E+09,8.999999E+09,8.999999E+09,8.999999E+09,8.999999E+09]];
	LOCAL CONST Robtarget Tr_meulage_motif_1_P110 :=[[-101.391265625,-74.2858203125,46.30380859375],[0.697372246118371,-0.704623915003405,0.0931525017095072,-0.0921938185257175],[0,0,0,0],[8.999999E+09,8.999999E+09,8.999999E+09,8.999999E+09,8.999999E+09,8.999999E+09]];
	LOCAL CONST Robtarget Tr_meulage_motif_1_P111 :=[[-102.3598125,-74.036984375,46.30380859375],[0.697372246118371,-0.704623915003405,0.0931525017095072,-0.0921938185257175],[0,0,0,0],[8.999999E+09,8.999999E+09,8.999999E+09,8.999999E+09,8.999999E+09,8.999999E+09]];
	LOCAL CONST Robtarget Tr_meulage_motif_1_P112 :=[[-103.328359375,-73.78815625,46.30380859375],[0.697372246118371,-0.704623915003405,0.0931525017095072,-0.0921938185257175],[0,0,0,0],[8.999999E+09,8.999999E+09,8.999999E+09,8.999999E+09,8.999999E+09,8.999999E+09]];
	LOCAL CONST Robtarget Tr_meulage_motif_1_P113 :=[[-104.29690625,-73.5393203125,46.30380859375],[0.697372246118371,-0.704623915003405,0.0931525017095072,-0.0921938185257175],[0,0,0,0],[8.999999E+09,8.999999E+09,8.999999E+09,8.999999E+09,8.999999E+09,8.999999E+09]];
	LOCAL CONST Robtarget Tr_meulage_motif_1_P114 :=[[-105.265453125,-73.2904921875,46.30380859375],[0.697372246118371,-0.704623915003405,0.0931525017095072,-0.0921938185257175],[0,0,0,0],[8.999999E+09,8.999999E+09,8.999999E+09,8.999999E+09,8.999999E+09,8.999999E+09]];
	LOCAL CONST Robtarget Tr_meulage_motif_1_P115 :=[[-106.234,-73.0416640625,46.30380859375],[0.697372246118371,-0.704623915003405,0.0931525017095072,-0.0921938185257175],[0,0,0,0],[8.999999E+09,8.999999E+09,8.999999E+09,8.999999E+09,8.999999E+09,8.999999E+09]];
	LOCAL CONST Robtarget Tr_meulage_motif_1_degg1 :=[[-108.832478773948,-82.6976056112364,46.4072535971393],[0.697372246118371,-0.704623915003405,0.0931525017095072,-0.0921938185257175],[0,0,0,0],[8.999999E+09,8.999999E+09,8.999999E+09,8.999999E+09,8.999999E+09,8.999999E+09]];
	LOCAL CONST Robtarget Tr_meulage_motif_1_degg2 :=[[-158.203575478964,-266.160495037229,48.372708661536],[0.697372246118371,-0.704623915003405,0.0931525017095072,-0.0921938185257175],[0,0,0,0],[8.999999E+09,8.999999E+09,8.999999E+09,8.999999E+09,8.999999E+09,8.999999E+09]];
	LOCAL CONST Robtarget Tr_meulage_bavure_App1 :=[[269.845469635261,-247.024526100345,47.4674132182396],[0.640300650580774,-0.632243257862969,-0.306491428807427,0.310397396606735],[0,0,0,0],[8.999999E+09,8.999999E+09,8.999999E+09,8.999999E+09,8.999999E+09,8.999999E+09]];
	LOCAL CONST Robtarget Tr_meulage_bavure_App2 :=[[120.698007075513,-129.341707555017,49.873370660912],[0.640300650580774,-0.632243257862969,-0.306491428807427,0.310397396606735],[0,0,0,0],[8.999999E+09,8.999999E+09,8.999999E+09,8.999999E+09,8.999999E+09,8.999999E+09]];
	LOCAL CONST Robtarget Tr_meulage_bavure_P0 :=[[112.848140625,-123.147875,50],[0.640300650580774,-0.632243257862969,-0.306491428807427,0.310397396606735],[0,0,0,0],[8.999999E+09,8.999999E+09,8.999999E+09,8.999999E+09,8.999999E+09,8.999999E+09]];
	LOCAL CONST Robtarget Tr_meulage_bavure_P1 :=[[112.11834375,-124.76703125,50],[0.645099448478915,-0.637031484332328,-0.296476838960431,0.300231699694721],[0,0,0,0],[8.999999E+09,8.999999E+09,8.999999E+09,8.999999E+09,8.999999E+09,8.999999E+09]];
	LOCAL CONST Robtarget Tr_meulage_bavure_P2 :=[[111.6141328125,-126.211453125,50],[0.658133973881904,-0.650042609034397,-0.266944974340852,0.270267755265642],[0,0,0,0],[8.999999E+09,8.999999E+09,8.999999E+09,8.999999E+09,8.999999E+09,8.999999E+09]];
	LOCAL CONST Robtarget Tr_meulage_bavure_P3 :=[[109.83325,-127.8506953125,50],[0.675463618715307,-0.667388351462461,-0.220407544637985,0.223074432400702],[0,0,0,0],[8.999999E+09,8.999999E+09,8.999999E+09,8.999999E+09,8.999999E+09,8.999999E+09]];
	LOCAL CONST Robtarget Tr_meulage_bavure_P4 :=[[107.33709375,-129.8155078125,50],[0.69182107672061,-0.683867279380433,-0.162923454464394,0.164818354509831],[0,0,0,0],[8.999999E+09,8.999999E+09,8.999999E+09,8.999999E+09,8.999999E+09,8.999999E+09]];
	LOCAL CONST Robtarget Tr_meulage_bavure_P5 :=[[105.6083671875,-130.0857578125,50],[0.703295752772457,-0.695601485357323,-0.103143115124797,0.104284013651476],[0,0,0,0],[8.999999E+09,8.999999E+09,8.999999E+09,8.999999E+09,8.999999E+09,8.999999E+09]];
	LOCAL CONST Robtarget Tr_meulage_bavure_P6 :=[[104.2345546875,-130.3357421875,50],[0.709063485911645,-0.701750554055035,-0.0486087981340681,0.0491153496805287],[0,0,0,0],[8.999999E+09,8.999999E+09,8.999999E+09,8.999999E+09,8.999999E+09,8.999999E+09]];
	LOCAL CONST Robtarget Tr_meulage_bavure_P7 :=[[103.3832734375,-130.186078125,50],[0.710518982215175,-0.703662093640687,-0.00333289224993684,0.00336536987093579],[0,0,0,0],[8.999999E+09,8.999999E+09,8.999999E+09,8.999999E+09,8.999999E+09,8.999999E+09]];
	LOCAL CONST Robtarget Tr_meulage_bavure_P8 :=[[100.108578125,-129.9469140625,50],[0.709556946720167,-0.703202425373939,0.0317567270726456,-0.0320436982103833],[0,0,0,0],[8.999999E+09,8.999999E+09,8.999999E+09,8.999999E+09,8.999999E+09,8.999999E+09]];
	LOCAL CONST Robtarget Tr_meulage_bavure_P9 :=[[97.5049453125,-129.101609375,50],[0.707678338761457,-0.701829309043884,0.0573236023022823,-0.0578013359179404],[0,0,0,0],[8.999999E+09,8.999999E+09,8.999999E+09,8.999999E+09,8.999999E+09,8.999999E+09]];
	LOCAL CONST Robtarget Tr_meulage_bavure_P10 :=[[96.9781171875,-128.9456015625,50],[0.705802450309124,-0.700432113954917,0.0746723621301829,-0.0752448882794166],[0,0,0,0],[8.999999E+09,8.999999E+09,8.999999E+09,8.999999E+09,8.999999E+09,8.999999E+09]];
	LOCAL CONST Robtarget Tr_meulage_bavure_P11 :=[[90.0638125,-127.106203125,50],[0.704347574657057,-0.69942210369198,0.0854401443253655,-0.0860418309862605],[0,0,0,0],[8.999999E+09,8.999999E+09,8.999999E+09,8.999999E+09,8.999999E+09,8.999999E+09]];
	LOCAL CONST Robtarget Tr_meulage_bavure_P12 :=[[85.2067890625,-125.6455390625,50],[0.703398247696666,-0.698871618997784,0.09138063999038,-0.0919725172626261],[0,0,0,0],[8.999999E+09,8.999999E+09,8.999999E+09,8.999999E+09,8.999999E+09,8.999999E+09]];
	LOCAL CONST Robtarget Tr_meulage_bavure_P13 :=[[82.11053125,-124.8009765625,50],[0.70285599921477,-0.698676773163084,0.0941748181999816,-0.0947381371319284],[0,0,0,0],[8.999999E+09,8.999999E+09,8.999999E+09,8.999999E+09,8.999999E+09,8.999999E+09]];
	LOCAL CONST Robtarget Tr_meulage_bavure_P14 :=[[74.224453125,-122.6573046875,50],[0.702571570449618,-0.698687551871477,0.0952046220444709,-0.0957338665111216],[0,0,0,0],[8.999999E+09,8.999999E+09,8.999999E+09,8.999999E+09,8.999999E+09,8.999999E+09]];
	LOCAL CONST Robtarget Tr_meulage_bavure_P15 :=[[69.749453125,-121.524703125,50],[0.702432944773348,-0.698787439630677,0.0953649173349673,-0.0958624267017052],[0,0,0,0],[8.999999E+09,8.999999E+09,8.999999E+09,8.999999E+09,8.999999E+09,8.999999E+09]];
	LOCAL CONST Robtarget Tr_meulage_bavure_P16 :=[[64.85916015625,-120.246671875,50],[0.702371170576915,-0.698921370255658,0.0951160498532654,-0.0955855323920816],[0,0,0,0],[8.999999E+09,8.999999E+09,8.999999E+09,8.999999E+09,8.999999E+09,8.999999E+09]];
	LOCAL CONST Robtarget Tr_meulage_bavure_P17 :=[[56.47085546875,-117.8733984375,50],[0.702364809384447,-0.699059462049067,0.0946431123228651,-0.0950906112497969],[0,0,0,0],[8.999999E+09,8.999999E+09,8.999999E+09,8.999999E+09,8.999999E+09,8.999999E+09]];
	LOCAL CONST Robtarget Tr_meulage_bavure_P18 :=[[54.4977734375,-117.3357265625,50],[0.70239812172387,-0.699198617527353,0.0940135551433683,-0.0944437573157845],[0,0,0,0],[8.999999E+09,8.999999E+09,8.999999E+09,8.999999E+09,8.999999E+09,8.999999E+09]];
	LOCAL CONST Robtarget Tr_meulage_bavure_P19 :=[[53.78018359375,-117.1455234375,50],[0.702453715119241,-0.699332488035347,0.0933138528716889,-0.0937303267662506],[0,0,0,0],[8.999999E+09,8.999999E+09,8.999999E+09,8.999999E+09,8.999999E+09,8.999999E+09]];
	LOCAL CONST Robtarget Tr_meulage_bavure_P20 :=[[50.9853515625,-116.481796875,50],[0.702512483913347,-0.699440652652299,0.0926912917169056,-0.093098377016342],[0,0,0,0],[8.999999E+09,8.999999E+09,8.999999E+09,8.999999E+09,8.999999E+09,8.999999E+09]];
	LOCAL CONST Robtarget Tr_meulage_bavure_P21 :=[[44.32946875,-114.892484375,50],[0.702548631271834,-0.699509583373495,0.0922972973706903,-0.0926982867413347],[0,0,0,0],[8.999999E+09,8.999999E+09,8.999999E+09,8.999999E+09,8.999999E+09,8.999999E+09]];
	LOCAL CONST Robtarget Tr_meulage_bavure_P22 :=[[40.29147265625,-113.757875,50],[0.702552456394782,-0.699529416907035,0.0922089867103777,-0.092607470893049],[0,0,0,0],[8.999999E+09,8.999999E+09,8.999999E+09,8.999999E+09,8.999999E+09,8.999999E+09]];
	LOCAL CONST Robtarget Tr_meulage_bavure_P23 :=[[39.119109375,-113.4477265625,50],[0.702525188855789,-0.699511630141392,0.0923800541727568,-0.0927780357148685],[0,0,0,0],[8.999999E+09,8.999999E+09,8.999999E+09,8.999999E+09,8.999999E+09,8.999999E+09]];
	LOCAL CONST Robtarget Tr_meulage_bavure_P24 :=[[37.37289453125,-112.9351171875,50],[0.702486660759462,-0.699474301460216,0.0926662609884627,-0.0930653379415863],[0,0,0,0],[8.999999E+09,8.999999E+09,8.999999E+09,8.999999E+09,8.999999E+09,8.999999E+09]];
	LOCAL CONST Robtarget Tr_meulage_bavure_P25 :=[[32.36602734375,-111.57046875,50],[0.702462794453206,-0.699437216002823,0.09289452329317,-0.0932963601720261],[0,0,0,0],[8.999999E+09,8.999999E+09,8.999999E+09,8.999999E+09,8.999999E+09,8.999999E+09]];
	LOCAL CONST Robtarget Tr_meulage_bavure_P26 :=[[23.438201171875,-109.0511796875,50],[0.70246347792942,-0.699420285283626,0.0929542178920436,-0.0933586636855623],[0,0,0,0],[8.999999E+09,8.999999E+09,8.999999E+09,8.999999E+09,8.999999E+09,8.999999E+09]];
	LOCAL CONST Robtarget Tr_meulage_bavure_P27 :=[[20.495330078125,-108.2079453125,50],[0.702495216310289,-0.699417774658647,0.0928418762967156,-0.0932503810094697],[0,0,0,0],[8.999999E+09,8.999999E+09,8.999999E+09,8.999999E+09,8.999999E+09,8.999999E+09]];
	LOCAL CONST Robtarget Tr_meulage_bavure_P28 :=[[13.812560546875,-106.439328125,50],[0.702547312368637,-0.699412927136009,0.0926598743819643,-0.0930751251310594],[0,0,0,0],[8.999999E+09,8.999999E+09,8.999999E+09,8.999999E+09,8.999999E+09,8.999999E+09]];
	LOCAL CONST Robtarget Tr_meulage_bavure_P29 :=[[5.49478125,-104.3263828125,50],[0.702601300245467,-0.699386437187952,0.092550248600471,-0.0929756734577012],[0,0,0,0],[8.999999E+09,8.999999E+09,8.999999E+09,8.999999E+09,8.999999E+09,8.999999E+09]];
	LOCAL CONST Robtarget Tr_meulage_bavure_P30 :=[[0.9022216796875,-103.1025703125,50],[0.702645173103038,-0.699323520059588,0.0926139836902965,-0.0930538824095111],[0,0,0,0],[8.999999E+09,8.999999E+09,8.999999E+09,8.999999E+09,8.999999E+09,8.999999E+09]];
	LOCAL CONST Robtarget Tr_meulage_bavure_P31 :=[[-0.019683837890625,-102.8685,50],[0.702676060282315,-0.699220842261638,0.0928738677334348,-0.0933328063720552],[0,0,0,0],[8.999999E+09,8.999999E+09,8.999999E+09,8.999999E+09,8.999999E+09,8.999999E+09]];
	LOCAL CONST Robtarget Tr_meulage_bavure_P32 :=[[-3.64862060546875,-101.858875,50],[0.702703134031038,-0.699081642991126,0.0932812301302015,-0.0937644600111394],[0,0,0,0],[8.999999E+09,8.999999E+09,8.999999E+09,8.999999E+09,8.999999E+09,8.999999E+09]];
	LOCAL CONST Robtarget Tr_meulage_bavure_P33 :=[[-8.565857421875,-100.5127265625,50],[0.702734272991826,-0.698915230333594,0.0937701641379621,-0.0942825471014029],[0,0,0,0],[8.999999E+09,8.999999E+09,8.999999E+09,8.999999E+09,8.999999E+09,8.999999E+09]];
	LOCAL CONST Robtarget Tr_meulage_bavure_P34 :=[[-12.509705078125,-99.4137890625,50],[0.702764643025494,-0.698731988761665,0.0943198832132003,-0.0948642399698985],[0,0,0,0],[8.999999E+09,8.999999E+09,8.999999E+09,8.999999E+09,8.999999E+09,8.999999E+09]];
	LOCAL CONST Robtarget Tr_meulage_bavure_P35 :=[[-16.4847109375,-98.3364140625,50],[0.702790630730192,-0.698523841756833,0.094971696578999,-0.0955518116209214],[0,0,0,0],[8.999999E+09,8.999999E+09,8.999999E+09,8.999999E+09,8.999999E+09,8.999999E+09]];
	LOCAL CONST Robtarget Tr_meulage_bavure_P36 :=[[-18.151611328125,-97.91784375,50],[0.70279095138542,-0.698288961418033,0.0958088252409874,-0.0964265213436812],[0,0,0,0],[8.999999E+09,8.999999E+09,8.999999E+09,8.999999E+09,8.999999E+09,8.999999E+09]];
	LOCAL CONST Robtarget Tr_meulage_bavure_P37 :=[[-20.977935546875,-97.0919375,50],[0.702750956791196,-0.698025040777814,0.096888062153251,-0.0975440340993653],[0,0,0,0],[8.999999E+09,8.999999E+09,8.999999E+09,8.999999E+09,8.999999E+09,8.999999E+09]];
	LOCAL CONST Robtarget Tr_meulage_bavure_P38 :=[[-25.68051171875,-95.8036640625,50],[0.702666003760366,-0.697741868967437,0.0981840772779468,-0.0988769862927826],[0,0,0,0],[8.999999E+09,8.999999E+09,8.999999E+09,8.999999E+09,8.999999E+09,8.999999E+09]];
	LOCAL CONST Robtarget Tr_meulage_bavure_P39 :=[[-27.627716796875,-95.237,50],[0.702546600461798,-0.697461986682963,0.0995739942374592,-0.100299905201469],[0,0,0,0],[8.999999E+09,8.999999E+09,8.999999E+09,8.999999E+09,8.999999E+09,8.999999E+09]];
	LOCAL CONST Robtarget Tr_meulage_bavure_P40 :=[[-30.55847265625,-94.366453125,50],[0.702408131949015,-0.697224041709529,0.100870172693789,-0.101620175628907],[0,0,0,0],[8.999999E+09,8.999999E+09,8.999999E+09,8.999999E+09,8.999999E+09,8.999999E+09]];
	LOCAL CONST Robtarget Tr_meulage_bavure_P41 :=[[-36.29049609375,-92.7145390625,50],[0.702268058321205,-0.697064407190405,0.101895028767073,-0.10265568470675],[0,0,0,0],[8.999999E+09,8.999999E+09,8.999999E+09,8.999999E+09,8.999999E+09,8.999999E+09]];
	LOCAL CONST Robtarget Tr_meulage_bavure_P42 :=[[-39.8259296875,-91.570875,50],[0.702139416566781,-0.697003152281906,0.102545827142686,-0.103301494413044],[0,0,0,0],[8.999999E+09,8.999999E+09,8.999999E+09,8.999999E+09,8.999999E+09,8.999999E+09]];
	LOCAL CONST Robtarget Tr_meulage_bavure_P43 :=[[-44.2456953125,-90.288375,50],[0.702013143708012,-0.697049986222412,0.102829348477008,-0.103561517275116],[0,0,0,0],[8.999999E+09,8.999999E+09,8.999999E+09,8.999999E+09,8.999999E+09,8.999999E+09]];
	LOCAL CONST Robtarget Tr_meulage_bavure_P44 :=[[-52.09060546875,-87.944609375,50],[0.701869175014875,-0.697197629290017,0.102841911999317,-0.10353100024941],[0,0,0,0],[8.999999E+09,8.999999E+09,8.999999E+09,8.999999E+09,8.999999E+09,8.999999E+09]];
	LOCAL CONST Robtarget Tr_meulage_bavure_P45 :=[[-52.18337890625,-87.9156171875,50],[0.701686786982292,-0.697430182719958,0.102707438167298,-0.103334289327325],[0,0,0,0],[8.999999E+09,8.999999E+09,8.999999E+09,8.999999E+09,8.999999E+09,8.999999E+09]];
	LOCAL CONST Robtarget Tr_meulage_bavure_P46 :=[[-52.21298046875,-87.9071953125,50],[0.701448353000857,-0.697734090300347,0.102530790262083,-0.103076594595307],[0,0,0,0],[8.999999E+09,8.999999E+09,8.999999E+09,8.999999E+09,8.999999E+09,8.999999E+09]];
	LOCAL CONST Robtarget Tr_meulage_bavure_P47 :=[[-52.25674609375,-87.896453125,50],[0.701146984657349,-0.698099032681869,0.102369278678357,-0.102816230515516],[0,0,0,0],[8.999999E+09,8.999999E+09,8.999999E+09,8.999999E+09,8.999999E+09,8.999999E+09]];
	LOCAL CONST Robtarget Tr_meulage_bavure_P48 :=[[-52.336609375,-87.872453125,50],[0.700779439150608,-0.698520333613109,0.102249173274606,-0.102579860389117],[0,0,0,0],[8.999999E+09,8.999999E+09,8.999999E+09,8.999999E+09,8.999999E+09,8.999999E+09]];
	LOCAL CONST Robtarget Tr_meulage_bavure_P49 :=[[-55.57409765625,-86.9306484375,50],[0.700345726130666,-0.69898982259128,0.102197193787602,-0.102395436354652],[0,0,0,0],[8.999999E+09,8.999999E+09,8.999999E+09,8.999999E+09,8.999999E+09,8.999999E+09]];
	LOCAL CONST Robtarget Tr_meulage_bavure_P50 :=[[-57.9013359375,-86.2210703125,50],[0.699850778940445,-0.69949069751899,0.102251855966129,-0.102304492825738],[0,0,0,0],[8.999999E+09,8.999999E+09,8.999999E+09,8.999999E+09,8.999999E+09,8.999999E+09]];
	LOCAL CONST Robtarget Tr_meulage_bavure_P51 :=[[-60.0220625,-85.6057734375,50],[0.699294408623828,-0.700010461648281,0.10245522912525,-0.10235042586772],[0,0,0,0],[8.999999E+09,8.999999E+09,8.999999E+09,8.999999E+09,8.999999E+09,8.999999E+09]];
	LOCAL CONST Robtarget Tr_meulage_bavure_P52 :=[[-66.7958671875,-83.662,50],[0.698688522880542,-0.700538761291948,0.102799661121138,-0.102528150260932],[0,0,0,0],[8.999999E+09,8.999999E+09,8.999999E+09,8.999999E+09,8.999999E+09,8.999999E+09]];
	LOCAL CONST Robtarget Tr_meulage_bavure_P53 :=[[-67.645078125,-83.4156640625,50],[0.698058291582974,-0.70107483089083,0.103199212200436,-0.102755173324091],[0,0,0,0],[8.999999E+09,8.999999E+09,8.999999E+09,8.999999E+09,8.999999E+09,8.999999E+09]];
	LOCAL CONST Robtarget Tr_meulage_bavure_P54 :=[[-68.705046875,-83.1078671875,50],[0.697439109645332,-0.701630205174809,0.103492315605252,-0.102874117902147],[0,0,0,0],[8.999999E+09,8.999999E+09,8.999999E+09,8.999999E+09,8.999999E+09,8.999999E+09]];
	LOCAL CONST Robtarget Tr_meulage_bavure_P55 :=[[-72.89453125,-81.7782890625,50],[0.696873771114332,-0.702219311430677,0.103482853737202,-0.102695105867416],[0,0,0,0],[8.999999E+09,8.999999E+09,8.999999E+09,8.999999E+09,8.999999E+09,8.999999E+09]];
	LOCAL CONST Robtarget Tr_meulage_bavure_P56 :=[[-74.2646484375,-81.33534375,50],[0.696397876865545,-0.702850952990912,0.103015796619059,-0.102069979052946],[0,0,0,0],[8.999999E+09,8.999999E+09,8.999999E+09,8.999999E+09,8.999999E+09,8.999999E+09]];
	LOCAL CONST Robtarget Tr_meulage_bavure_P57 :=[[-76.1800859375,-80.7783046875,50],[0.696032763961537,-0.703515669574791,0.102040222242215,-0.100954877046911],[0,0,0,0],[8.999999E+09,8.999999E+09,8.999999E+09,8.999999E+09,8.999999E+09,8.999999E+09]];
	LOCAL CONST Robtarget Tr_meulage_bavure_P58 :=[[-78.376984375,-80.1273671875,50],[0.695777286283564,-0.704189188648134,0.100628103622797,-0.0994260491231644],[0,0,0,0],[8.999999E+09,8.999999E+09,8.999999E+09,8.999999E+09,8.999999E+09,8.999999E+09]];
	LOCAL CONST Robtarget Tr_meulage_bavure_P59 :=[[-79.144625,-79.927828125,50],[0.695615434675039,-0.704832556240526,0.0989562266402808,-0.097662172382245],[0,0,0,0],[8.999999E+09,8.999999E+09,8.999999E+09,8.999999E+09,8.999999E+09,8.999999E+09]];
	LOCAL CONST Robtarget Tr_meulage_bavure_P60 :=[[-82.3830234375,-79.06440625,50],[0.695526908788096,-0.705399567824242,0.097253973746672,-0.0958928227529555],[0,0,0,0],[8.999999E+09,8.999999E+09,8.999999E+09,8.999999E+09,8.999999E+09,8.999999E+09]];
	LOCAL CONST Robtarget Tr_meulage_bavure_P61 :=[[-82.549625,-79.0198984375,50],[0.695491837463084,-0.705849432165929,0.0957464158365789,-0.0943414383381311],[0,0,0,0],[8.999999E+09,8.999999E+09,8.999999E+09,8.999999E+09,8.999999E+09,8.999999E+09]];
	LOCAL CONST Robtarget Tr_meulage_bavure_P62 :=[[-82.7827734375,-78.95759375,50],[0.695495082444396,-0.706154041438152,0.0946076866149303,-0.093179642034078],[0,0,0,0],[8.999999E+09,8.999999E+09,8.999999E+09,8.999999E+09,8.999999E+09,8.999999E+09]];
	LOCAL CONST Robtarget Tr_meulage_bavure_P63 :=[[-93.2647421875,-76.2340390625,50],[0.695530186076176,-0.706298911909447,0.0939324457143587,-0.092500286131935],[0,0,0,0],[8.999999E+09,8.999999E+09,8.999999E+09,8.999999E+09,8.999999E+09,8.999999E+09]];
	LOCAL CONST Robtarget Tr_meulage_bavure_P64 :=[[-99.5831015625,-74.5251640625,50],[0.695603285936978,-0.706276618333315,0.0937362390141461,-0.0923196863340625],[0,0,0,0],[8.999999E+09,8.999999E+09,8.999999E+09,8.999999E+09,8.999999E+09,8.999999E+09]];
	LOCAL CONST Robtarget Tr_meulage_bavure_P65 :=[[-101.133453125,-74.125125,50],[0.695723100422288,-0.706093177533342,0.0939660606594633,-0.0925860228317863],[0,0,0,0],[8.999999E+09,8.999999E+09,8.999999E+09,8.999999E+09,8.999999E+09,8.999999E+09]];
	LOCAL CONST Robtarget Tr_meulage_bavure_P66 :=[[-104.3062109375,-73.3186484375,50],[0.695895403592743,-0.705765774474219,0.0945316438965455,-0.0932095871759718],[0,0,0,0],[8.999999E+09,8.999999E+09,8.999999E+09,8.999999E+09,8.999999E+09,8.999999E+09]];
	LOCAL CONST Robtarget Tr_meulage_bavure_P67 :=[[-109.7843359375,-71.7966484375,50],[0.696129072432796,-0.705314319414796,0.0953182182211366,-0.0940768973629811],[0,0,0,0],[8.999999E+09,8.999999E+09,8.999999E+09,8.999999E+09,8.999999E+09,8.999999E+09]];
	LOCAL CONST Robtarget Tr_meulage_bavure_P68 :=[[-115.1020234375,-70.3434765625,50],[0.696438663177283,-0.704757169540365,0.0961968921822461,-0.0950614451171973],[0,0,0,0],[8.999999E+09,8.999999E+09,8.999999E+09,8.999999E+09,8.999999E+09,8.999999E+09]];
	LOCAL CONST Robtarget Tr_meulage_bavure_P69 :=[[-115.1598828125,-70.361390625,50],[0.696832057177351,-0.70412414889358,0.0970264076154568,-0.0960215770549087],[0,0,0,0],[8.999999E+09,8.999999E+09,8.999999E+09,8.999999E+09,8.999999E+09,8.999999E+09]];
	LOCAL CONST Robtarget Tr_meulage_bavure_P70 :=[[-123.5550859375,-67.8595703125,50],[0.697309905961321,-0.703444711026951,0.0976990146332908,-0.0968469726739386],[0,0,0,0],[8.999999E+09,8.999999E+09,8.999999E+09,8.999999E+09,8.999999E+09,8.999999E+09]];
	LOCAL CONST Robtarget Tr_meulage_bavure_P71 :=[[-125.9613984375,-67.190859375,50],[0.697864752518907,-0.702737278370125,0.0981791989118959,-0.0974984598939521],[0,0,0,0],[8.999999E+09,8.999999E+09,8.999999E+09,8.999999E+09,8.999999E+09,8.999999E+09]];
	LOCAL CONST Robtarget Tr_meulage_bavure_P72 :=[[-126.8297734375,-66.96953125,50],[0.698467404080317,-0.701998890515341,0.0985859630556769,-0.0980900149909168],[0,0,0,0],[8.999999E+09,8.999999E+09,8.999999E+09,8.999999E+09,8.999999E+09,8.999999E+09]];
	LOCAL CONST Robtarget Tr_meulage_bavure_P73 :=[[-135.4400625,-64.56103515625,50],[0.699046797974772,-0.701190110831529,0.0993131593406462,-0.0990095909246462],[0,0,0,0],[8.999999E+09,8.999999E+09,8.999999E+09,8.999999E+09,8.999999E+09,8.999999E+09]];
	LOCAL CONST Robtarget Tr_meulage_bavure_P74 :=[[-139.74225,-63.282578125,50],[0.699489685270955,-0.700231332076267,0.101024426420803,-0.100917426862684],[0,0,0,0],[8.999999E+09,8.999999E+09,8.999999E+09,8.999999E+09,8.999999E+09,8.999999E+09]];
	LOCAL CONST Robtarget Tr_meulage_bavure_P75 :=[[-145.268125,-61.800046875,50],[0.699638865939984,-0.698996694886196,0.104615866609625,-0.104711977623876],[0,0,0,0],[8.999999E+09,8.999999E+09,8.999999E+09,8.999999E+09,8.999999E+09,8.999999E+09]];
	LOCAL CONST Robtarget Tr_meulage_bavure_P76 :=[[-145.89440625,-61.638703125,50],[0.699289586216509,-0.697315310871415,0.111075358338495,-0.111389840665208],[0,0,0,0],[8.999999E+09,8.999999E+09,8.999999E+09,8.999999E+09,8.999999E+09,8.999999E+09]];
	LOCAL CONST Robtarget Tr_meulage_bavure_P77 :=[[-148.015203125,-61.17715625,50],[0.69817848448718,-0.694956591374478,0.121336952011691,-0.121899483103352],[0,0,0,0],[8.999999E+09,8.999999E+09,8.999999E+09,8.999999E+09,8.999999E+09,8.999999E+09]];
	LOCAL CONST Robtarget Tr_meulage_bavure_P78 :=[[-150.214484375,-60.7230546875,50],[0.695981999672108,-0.691626727556321,0.1360654686003,-0.136922292256335],[0,0,0,0],[8.999999E+09,8.999999E+09,8.999999E+09,8.999999E+09,8.999999E+09,8.999999E+09]];
	LOCAL CONST Robtarget Tr_meulage_bavure_P79 :=[[-150.357078125,-60.6689296875,50],[0.6922950746234,-0.686944420458,0.155653454973361,-0.156865849720896],[0,0,0,0],[8.999999E+09,8.999999E+09,8.999999E+09,8.999999E+09,8.999999E+09,8.999999E+09]];
	LOCAL CONST Robtarget Tr_meulage_bavure_P80 :=[[-154.13815625,-59.23426953125,50],[0.686588283837594,-0.680408367600724,0.180343414958798,-0.181981412448815],[0,0,0,0],[8.999999E+09,8.999999E+09,8.999999E+09,8.999999E+09,8.999999E+09,8.999999E+09]];
	LOCAL CONST Robtarget Tr_meulage_bavure_P81 :=[[-156.4303125,-57.36402734375,50],[0.678146032171779,-0.671326208891954,0.210398559214684,-0.212535941865873],[0,0,0,0],[8.999999E+09,8.999999E+09,8.999999E+09,8.999999E+09,8.999999E+09,8.999999E+09]];
	LOCAL CONST Robtarget Tr_meulage_bavure_P82 :=[[-156.664046875,-57.19488671875,50],[0.665968964473117,-0.658719978157345,0.246203039197499,-0.248912418784007],[0,0,0,0],[8.999999E+09,8.999999E+09,8.999999E+09,8.999999E+09,8.999999E+09,8.999999E+09]];
	LOCAL CONST Robtarget Tr_meulage_bavure_P83 :=[[-156.845125,-56.74064453125,50],[0.648799463103432,-0.641347209718396,0.287919546857203,-0.291265081670751],[0,0,0,0],[8.999999E+09,8.999999E+09,8.999999E+09,8.999999E+09,8.999999E+09,8.999999E+09]];
	LOCAL CONST Robtarget Tr_meulage_bavure_P84 :=[[-157.411125,-55.2014140625,50],[0.625490341886798,-0.618069612698895,0.334698131312597,-0.338716617484927],[0,0,0,0],[8.999999E+09,8.999999E+09,8.999999E+09,8.999999E+09,8.999999E+09,8.999999E+09]];
	LOCAL CONST Robtarget Tr_meulage_bavure_P85 :=[[-157.667125,-54.40733203125,50],[0.595990095080112,-0.588825870676957,0.383715541820857,-0.388384195807514],[0,0,0,0],[8.999999E+09,8.999999E+09,8.999999E+09,8.999999E+09,8.999999E+09,8.999999E+09]];
	LOCAL CONST Robtarget Tr_meulage_bavure_P86 :=[[-157.728265625,-53.4144609375,50],[0.562353334370576,-0.555621669978148,0.430422439948145,-0.435637246297967],[0,0,0,0],[8.999999E+09,8.999999E+09,8.999999E+09,8.999999E+09,8.999999E+09,8.999999E+09]];
	LOCAL CONST Robtarget Tr_meulage_bavure_P87 :=[[-157.75390625,-51.0602734375,50],[0.528518619098751,-0.52231884956975,0.47040768273541,-0.47599128214032],[0,0,0,0],[8.999999E+09,8.999999E+09,8.999999E+09,8.999999E+09,8.999999E+09,8.999999E+09]];
	LOCAL CONST Robtarget Tr_meulage_bavure_P88 :=[[-157.40009375,-49.58351171875,50],[0.498492083186987,-0.49284974995614,0.501405720131149,-0.507146005394731],[0,0,0,0],[8.999999E+09,8.999999E+09,8.999999E+09,8.999999E+09,8.999999E+09,8.999999E+09]];
	LOCAL CONST Robtarget Tr_meulage_bavure_P89 :=[[-156.859984375,-47.4025859375,50],[0.474642723291579,-0.469539528663273,0.523572254691053,-0.529262704492535],[0,0,0,0],[8.999999E+09,8.999999E+09,8.999999E+09,8.999999E+09,8.999999E+09,8.999999E+09]];
	LOCAL CONST Robtarget Tr_meulage_bavure_P90 :=[[-156.85775,-47.3948359375,50],[0.457355793386055,-0.452758652189838,0.538478006501326,-0.543945509805726],[0,0,0,0],[8.999999E+09,8.999999E+09,8.999999E+09,8.999999E+09,8.999999E+09,8.999999E+09]];
	LOCAL CONST Robtarget Tr_meulage_bavure_P91 :=[[-155.977421875,-44.10205078125,50],[0.445728148616935,-0.441609842476495,0.548032530809578,-0.553143299455804],[0,0,0,0],[8.999999E+09,8.999999E+09,8.999999E+09,8.999999E+09,8.999999E+09,8.999999E+09]];
	LOCAL CONST Robtarget Tr_meulage_bavure_P92 :=[[-153.764265625,-35.87109375,50],[0.438325817994872,-0.434672986477405,0.553963206187832,-0.558618508730276],[0,0,0,0],[8.999999E+09,8.999999E+09,8.999999E+09,8.999999E+09,8.999999E+09,8.999999E+09]];
	LOCAL CONST Robtarget Tr_meulage_bavure_P93 :=[[-152.340546875,-30.861115234375,50],[0.433757747402881,-0.430569210437225,0.557603053204893,-0.561732326511502],[0,0,0,0],[8.999999E+09,8.999999E+09,8.999999E+09,8.999999E+09,8.999999E+09,8.999999E+09]];
	LOCAL CONST Robtarget Tr_meulage_bavure_P94 :=[[-150.999140625,-25.819611328125,50],[0.430931939566248,-0.428213501289732,0.559883121865609,-0.56343744162496],[0,0,0,0],[8.999999E+09,8.999999E+09,8.999999E+09,8.999999E+09,8.999999E+09,8.999999E+09]];
	LOCAL CONST Robtarget Tr_meulage_bavure_P95 :=[[-150.116609375,-22.5582890625,50],[0.42912881032316,-0.426890191143339,0.561381894363707,-0.564325790246067],[0,0,0,0],[8.999999E+09,8.999999E+09,8.999999E+09,8.999999E+09,8.999999E+09,8.999999E+09]];
	LOCAL CONST Robtarget Tr_meulage_bavure_P96 :=[[-148.586125,-17.323546875,50],[0.427959951258911,-0.426208229116008,0.562401779013977,-0.564713258666893],[0,0,0,0],[8.999999E+09,8.999999E+09,8.999999E+09,8.999999E+09,8.999999E+09,8.999999E+09]];
	LOCAL CONST Robtarget Tr_meulage_bavure_P97 :=[[-147.71325,-14.18490625,50],[0.427185418601868,-0.425925000303183,0.563125615382422,-0.564792044518024],[0,0,0,0],[8.999999E+09,8.999999E+09,8.999999E+09,8.999999E+09,8.999999E+09,8.999999E+09]];
	LOCAL CONST Robtarget Tr_meulage_bavure_P98 :=[[-146.710984375,-10.807037109375,50],[0.426681109175027,-0.425915982441893,0.563647203013559,-0.564659753753283],[0,0,0,0],[8.999999E+09,8.999999E+09,8.999999E+09,8.999999E+09,8.999999E+09,8.999999E+09]];
	LOCAL CONST Robtarget Tr_meulage_bavure_P99 :=[[-145.859296875,-7.934478515625,50],[0.426347406283627,-0.426078183425802,0.564040379878946,-0.564396775885376],[0,0,0,0],[8.999999E+09,8.999999E+09,8.999999E+09,8.999999E+09,8.999999E+09,8.999999E+09]];
	LOCAL CONST Robtarget Tr_meulage_bavure_P100 :=[[-145.327203125,-5.9014892578125,50],[0.426096124502709,-0.426319496988247,0.564370209098026,-0.564074504169538],[0,0,0,0],[8.999999E+09,8.999999E+09,8.999999E+09,8.999999E+09,8.999999E+09,8.999999E+09]];
	LOCAL CONST Robtarget Tr_meulage_bavure_P101 :=[[-144.324640625,-2.10446166992188,50],[0.425874910867974,-0.426581430983105,0.56467431959862,-0.563739084878312],[0,0,0,0],[8.999999E+09,8.999999E+09,8.999999E+09,8.999999E+09,8.999999E+09,8.999999E+09]];
	LOCAL CONST Robtarget Tr_meulage_bavure_P102 :=[[-142.352515625,5.1926572265625,50],[0.425654074849623,-0.426832681429707,0.564974699089892,-0.563414643061151],[0,0,0,0],[8.999999E+09,8.999999E+09,8.999999E+09,8.999999E+09,8.999999E+09,8.999999E+09]];
	LOCAL CONST Robtarget Tr_meulage_bavure_P103 :=[[-140.51321875,11.2269287109375,50],[0.425430516589332,-0.427069751513346,0.565273629177917,-0.563103922072019],[0,0,0,0],[8.999999E+09,8.999999E+09,8.999999E+09,8.999999E+09,8.999999E+09,8.999999E+09]];
	LOCAL CONST Robtarget Tr_meulage_bavure_P104 :=[[-138.51440625,17.958740234375,50],[0.425201396438565,-0.427281084201084,0.565570886040329,-0.56281810597581],[0,0,0,0],[8.999999E+09,8.999999E+09,8.999999E+09,8.999999E+09,8.999999E+09,8.999999E+09]];
	LOCAL CONST Robtarget Tr_meulage_bavure_P105 :=[[-136.483640625,25.252228515625,50],[0.424942011919126,-0.427439434343847,0.56588465259375,-0.562578329153184],[0,0,0,0],[8.999999E+09,8.999999E+09,8.999999E+09,8.999999E+09,8.999999E+09,8.999999E+09]];
	LOCAL CONST Robtarget Tr_meulage_bavure_P106 :=[[-135.08225,30.14367578125,50],[0.424611173670441,-0.427501606345889,0.566245896359713,-0.562417382929866],[0,0,0,0],[8.999999E+09,8.999999E+09,8.999999E+09,8.999999E+09,8.999999E+09,8.999999E+09]];
	LOCAL CONST Robtarget Tr_meulage_bavure_P107 :=[[-133.8308125,34.86468359375,50],[0.424163551740825,-0.427417956079771,0.566688128987361,-0.562373307207946],[0,0,0,0],[8.999999E+09,8.999999E+09,8.999999E+09,8.999999E+09,8.999999E+09,8.999999E+09]];
	LOCAL CONST Robtarget Tr_meulage_bavure_P108 :=[[-132.6279375,38.95388671875,50],[0.423584127612856,-0.427170282701718,0.567221949014143,-0.562460040329611],[0,0,0,0],[8.999999E+09,8.999999E+09,8.999999E+09,8.999999E+09,8.999999E+09,8.999999E+09]];
	LOCAL CONST Robtarget Tr_meulage_bavure_P109 :=[[-131.954984375,41.40908984375,50],[0.422913573868365,-0.426797436779964,0.567815689256773,-0.562648558186899],[0,0,0,0],[8.999999E+09,8.999999E+09,8.999999E+09,8.999999E+09,8.999999E+09,8.999999E+09]];
	LOCAL CONST Robtarget Tr_meulage_bavure_P110 :=[[-129.5341171875,50.724,50],[0.42225341235898,-0.426402270874319,0.568392231086519,-0.562861822106377],[0,0,0,0],[8.999999E+09,8.999999E+09,8.999999E+09,8.999999E+09,8.999999E+09,8.999999E+09]];
	LOCAL CONST Robtarget Tr_meulage_bavure_P111 :=[[-129.45321875,51.0257890625,50],[0.421744293428195,-0.426126951115243,0.568845055059352,-0.562994561100286],[0,0,0,0],[8.999999E+09,8.999999E+09,8.999999E+09,8.999999E+09,8.999999E+09,8.999999E+09]];
	LOCAL CONST Robtarget Tr_meulage_bavure_P112 :=[[-127.9983828125,56.07171484375,50],[0.421512448400378,-0.426096914104469,0.569078169220986,-0.56295533832646],[0,0,0,0],[8.999999E+09,8.999999E+09,8.999999E+09,8.999999E+09,8.999999E+09,8.999999E+09]];
	LOCAL CONST Robtarget Tr_meulage_bavure_P113 :=[[-126.818203125,59.814484375,50],[0.421614349125383,-0.426375200870522,0.569050342477936,-0.562696398086877],[0,0,0,0],[8.999999E+09,8.999999E+09,8.999999E+09,8.999999E+09,8.999999E+09,8.999999E+09]];
	LOCAL CONST Robtarget Tr_meulage_bavure_P114 :=[[-126.0251171875,62.442078125,50],[0.422008035523336,-0.426922436524432,0.56879343479616,-0.562245924554873],[0,0,0,0],[8.999999E+09,8.999999E+09,8.999999E+09,8.999999E+09,8.999999E+09,8.999999E+09]];
	LOCAL CONST Robtarget Tr_meulage_bavure_P115 :=[[-124.77225,66.809359375,50],[0.422562425650876,-0.427610533960611,0.56840721726333,-0.561696949463789],[0,0,0,0],[8.999999E+09,8.999999E+09,8.999999E+09,8.999999E+09,8.999999E+09,8.999999E+09]];
	LOCAL CONST Robtarget Tr_meulage_bavure_P116 :=[[-123.2723359375,72.3988671875,50],[0.423124062493638,-0.428287855384035,0.568009036807352,-0.561160649702569],[0,0,0,0],[8.999999E+09,8.999999E+09,8.999999E+09,8.999999E+09,8.999999E+09,8.999999E+09]];
	LOCAL CONST Robtarget Tr_meulage_bavure_P117 :=[[-120.677609375,81.3591640625,50],[0.423572330203497,-0.428840276694498,0.567693424282489,-0.560719782241529],[0,0,0,0],[8.999999E+09,8.999999E+09,8.999999E+09,8.999999E+09,8.999999E+09,8.999999E+09]];
	LOCAL CONST Robtarget Tr_meulage_bavure_P118 :=[[-119.8094140625,84.5329296875,50],[0.423875568688128,-0.429244587173381,0.567487643801137,-0.560389472407096],[0,0,0,0],[8.999999E+09,8.999999E+09,8.999999E+09,8.999999E+09,8.999999E+09,8.999999E+09]];
	LOCAL CONST Robtarget Tr_meulage_bavure_P119 :=[[-119.587921875,85.26440625,50],[0.424101794745449,-0.429573211282376,0.567341028731749,-0.560114881930338],[0,0,0,0],[8.999999E+09,8.999999E+09,8.999999E+09,8.999999E+09,8.999999E+09,8.999999E+09]];
	LOCAL CONST Robtarget Tr_meulage_bavure_P120 :=[[-114.8285546875,102.17309375,50],[0.424380769350738,-0.429964265398016,0.567155941944404,-0.55979088113614],[0,0,0,0],[8.999999E+09,8.999999E+09,8.999999E+09,8.999999E+09,8.999999E+09,8.999999E+09]];
	LOCAL CONST Robtarget Tr_meulage_bavure_P121 :=[[-114.11084375,104.69528125,50],[0.424864325922498,-0.430583201039999,0.566818358762541,-0.55929004971509],[0,0,0,0],[8.999999E+09,8.999999E+09,8.999999E+09,8.999999E+09,8.999999E+09,8.999999E+09]];
	LOCAL CONST Robtarget Tr_meulage_bavure_P122 :=[[-113.5258203125,106.8993828125,50],[0.425684670731983,-0.431571053184527,0.566226672224042,-0.558503664105338],[0,0,0,0],[8.999999E+09,8.999999E+09,8.999999E+09,8.999999E+09,8.999999E+09,8.999999E+09]];
	LOCAL CONST Robtarget Tr_meulage_bavure_P123 :=[[-112.61965625,109.940640625,50],[0.426892320677334,-0.432982401850219,0.565339195429529,-0.557387459803169],[0,0,0,0],[8.999999E+09,8.999999E+09,8.999999E+09,8.999999E+09,8.999999E+09,8.999999E+09]];
	LOCAL CONST Robtarget Tr_meulage_bavure_P124 :=[[-110.83603125,116.0145234375,50],[0.428424146584144,-0.434757595663988,0.564200999442121,-0.555981848502834],[0,0,0,0],[8.999999E+09,8.999999E+09,8.999999E+09,8.999999E+09,8.999999E+09,8.999999E+09]];
	LOCAL CONST Robtarget Tr_meulage_bavure_P125 :=[[-110.4515703125,117.3948359375,50],[0.430022776760754,-0.436646506404451,0.563011655249332,-0.554471023557738],[0,0,0,0],[8.999999E+09,8.999999E+09,8.999999E+09,8.999999E+09,8.999999E+09,8.999999E+09]];
	LOCAL CONST Robtarget Tr_meulage_bavure_P126 :=[[-109.9737890625,119.014921875,50],[0.431160295910903,-0.438116766338816,0.562188384321724,-0.55326188990077],[0,0,0,0],[8.999999E+09,8.999999E+09,8.999999E+09,8.999999E+09,8.999999E+09,8.999999E+09]];
	LOCAL CONST Robtarget Tr_meulage_bavure_P127 :=[[-109.7828984375,119.7498203125,50],[0.431066256931085,-0.438381399014187,0.562347494290316,-0.552963766262484],[0,0,0,0],[8.999999E+09,8.999999E+09,8.999999E+09,8.999999E+09,8.999999E+09,8.999999E+09]];
	LOCAL CONST Robtarget Tr_meulage_bavure_P128 :=[[-109.0510859375,122.644625,50],[0.428698775594594,-0.436381954404613,0.564315114180702,-0.554379474350311],[0,0,0,0],[8.999999E+09,8.999999E+09,8.999999E+09,8.999999E+09,8.999999E+09,8.999999E+09]];
	LOCAL CONST Robtarget Tr_meulage_bavure_P129 :=[[-108.5926171875,124.6397109375,50],[0.422886032093163,-0.430916716140854,0.568960223121194,-0.558356921795337],[0,0,0,0],[8.999999E+09,8.999999E+09,8.999999E+09,8.999999E+09,8.999999E+09,8.999999E+09]];
	LOCAL CONST Robtarget Tr_meulage_bavure_P130 :=[[-108.2261640625,126.749296875,50],[0.412431199831233,-0.420753194246914,0.577021604127385,-0.565608807663961],[0,0,0,0],[8.999999E+09,8.999999E+09,8.999999E+09,8.999999E+09,8.999999E+09,8.999999E+09]];
	LOCAL CONST Robtarget Tr_meulage_bavure_P131 :=[[-107.8736875,128.417296875,50],[0.396195255158859,-0.404706016794201,0.588929809484999,-0.576544915214887],[0,0,0,0],[8.999999E+09,8.999999E+09,8.999999E+09,8.999999E+09,8.999999E+09,8.999999E+09]];
	LOCAL CONST Robtarget Tr_meulage_bavure_P132 :=[[-107.818265625,128.697359375,50],[0.373278542330475,-0.381821739708786,0.604586388745404,-0.591058869711963],[0,0,0,0],[8.999999E+09,8.999999E+09,8.999999E+09,8.999999E+09,8.999999E+09,8.999999E+09]];
	LOCAL CONST Robtarget Tr_meulage_bavure_P133 :=[[-107.7569296875,128.8765546875,50],[0.343147436732221,-0.351519270573825,0.623284875325355,-0.608440632494255],[0,0,0,0],[8.999999E+09,8.999999E+09,8.999999E+09,8.999999E+09,8.999999E+09,8.999999E+09]];
	LOCAL CONST Robtarget Tr_meulage_bavure_P134 :=[[-106.754484375,131.849359375,50],[0.305865705818624,-0.313819068589111,0.643700247223662,-0.627386447030962],[0,0,0,0],[8.999999E+09,8.999999E+09,8.999999E+09,8.999999E+09,8.999999E+09,8.999999E+09]];
	LOCAL CONST Robtarget Tr_meulage_bavure_P135 :=[[-105.6456015625,133.20159375,50],[0.262272617564561,-0.269534645743521,0.664081248781751,-0.646189015564501],[0,0,0,0],[8.999999E+09,8.999999E+09,8.999999E+09,8.999999E+09,8.999999E+09,8.999999E+09]];
	LOCAL CONST Robtarget Tr_meulage_bavure_P136 :=[[-104.94653125,134.10146875,50],[0.213979571146591,-0.220281524264547,0.682630861803516,-0.663101726519391],[0,0,0,0],[8.999999E+09,8.999999E+09,8.999999E+09,8.999999E+09,8.999999E+09,8.999999E+09]];
	LOCAL CONST Robtarget Tr_meulage_bavure_P137 :=[[-103.763,134.617640625,50],[0.163259930335226,-0.168366795935664,0.69788853709131,-0.676720331429348],[0,0,0,0],[8.999999E+09,8.999999E+09,8.999999E+09,8.999999E+09,8.999999E+09,8.999999E+09]];
	LOCAL CONST Robtarget Tr_meulage_bavure_P138 :=[[-101.5198359375,135.8175625,50],[0.112777502196149,-0.116518098881147,0.709036400857749,-0.68627410696471],[0,0,0,0],[8.999999E+09,8.999999E+09,8.999999E+09,8.999999E+09,8.999999E+09,8.999999E+09]];
	LOCAL CONST Robtarget Tr_meulage_bavure_P139 :=[[-99.69528125,135.655359375,50],[0.0652600442470066,-0.0675503488395543,0.716014485461691,-0.691737908174449],[0,0,0,0],[8.999999E+09,8.999999E+09,8.999999E+09,8.999999E+09,8.999999E+09,8.999999E+09]];
	LOCAL CONST Robtarget Tr_meulage_bavure_P140 :=[[-96.8513515625,135.30609375,50],[0.0231360759404615,-0.0239934684515249,0.719451559039264,-0.693742379891639],[0,0,0,0],[8.999999E+09,8.999999E+09,8.999999E+09,8.999999E+09,8.999999E+09,8.999999E+09]];
	LOCAL CONST Robtarget Tr_meulage_bavure_P141 :=[[-96.6384609375,135.26559375,50],[0.0119543720168958,-0.0124212474618075,-0.720411039871427,0.693333065151622],[0,0,0,0],[8.999999E+09,8.999999E+09,8.999999E+09,8.999999E+09,8.999999E+09,8.999999E+09]];
	LOCAL CONST Robtarget Tr_meulage_bavure_P142 :=[[-94.722625,134.928046875,50],[0.0393066041742096,-0.0409209713126044,-0.720027552948801,0.691621853305466],[0,0,0,0],[8.999999E+09,8.999999E+09,8.999999E+09,8.999999E+09,8.999999E+09,8.999999E+09]];
	LOCAL CONST Robtarget Tr_meulage_bavure_P143 :=[[-88.7886328125,133.134578125,50],[0.0590868638256094,-0.0616334400247363,-0.719226516498429,0.689509448491829],[0,0,0,0],[8.999999E+09,8.999999E+09,8.999999E+09,8.999999E+09,8.999999E+09,8.999999E+09]];
	LOCAL CONST Robtarget Tr_meulage_bavure_P144 :=[[-86.786625,132.57275,50],[0.0721170872140994,-0.0753715664810032,-0.718591922963987,0.687563743189585],[0,0,0,0],[8.999999E+09,8.999999E+09,8.999999E+09,8.999999E+09,8.999999E+09,8.999999E+09]];
	LOCAL CONST Robtarget Tr_meulage_bavure_P145 :=[[-85.0901796875,132.104578125,50],[0.0794206222197151,-0.0831655132877919,-0.718404174798135,0.686054883954937],[0,0,0,0],[8.999999E+09,8.999999E+09,8.999999E+09,8.999999E+09,8.999999E+09,8.999999E+09]];
	LOCAL CONST Robtarget Tr_meulage_bavure_P146 :=[[-72.38290625,128.7671171875,50],[0.0818931260554111,-0.0859198045417954,-0.718748233184406,0.685063705349121],[0,0,0,0],[8.999999E+09,8.999999E+09,8.999999E+09,8.999999E+09,8.999999E+09,8.999999E+09]];
	LOCAL CONST Robtarget Tr_meulage_bavure_P147 :=[[-70.2894921875,128.1695546875,50],[0.0798823259705232,-0.0839694618486064,-0.719637215364092,0.684609539619052],[0,0,0,0],[8.999999E+09,8.999999E+09,8.999999E+09,8.999999E+09,8.999999E+09,8.999999E+09]];
	LOCAL CONST Robtarget Tr_meulage_bavure_P148 :=[[-64.38131640625,126.2659296875,50],[0.0729259941012189,-0.0768009106906184,-0.721085427162664,0.684703750709078],[0,0,0,0],[8.999999E+09,8.999999E+09,8.999999E+09,8.999999E+09,8.999999E+09,8.999999E+09]];
	LOCAL CONST Robtarget Tr_meulage_bavure_P149 :=[[-63.3453359375,125.9359140625,50],[0.0598241425500802,-0.0631192259091709,-0.723047965469229,0.685301885974045],[0,0,0,0],[8.999999E+09,8.999999E+09,8.999999E+09,8.999999E+09,8.999999E+09,8.999999E+09]];
	LOCAL CONST Robtarget Tr_meulage_bavure_P150 :=[[-62.654265625,125.7549453125,50],[0.0389622614683912,-0.04118261875078,-0.725249638318968,0.686147867600201],[0,0,0,0],[8.999999E+09,8.999999E+09,8.999999E+09,8.999999E+09,8.999999E+09,8.999999E+09]];
	LOCAL CONST Robtarget Tr_meulage_bavure_P151 :=[[-59.79998828125,124.9705234375,50],[0.0092189515054367,-0.0097615748891699,-0.72695927806678,0.686549292200822],[0,0,0,0],[8.999999E+09,8.999999E+09,8.999999E+09,8.999999E+09,8.999999E+09,8.999999E+09]];
	LOCAL CONST Robtarget Tr_meulage_bavure_P152 :=[[-58.43405078125,124.8461015625,50],[0.0289827035887404,-0.0307418897775627,0.726969307989098,-0.685368925723543],[0,0,0,0],[8.999999E+09,8.999999E+09,8.999999E+09,8.999999E+09,8.999999E+09,8.999999E+09]];
	LOCAL CONST Robtarget Tr_meulage_bavure_P153 :=[[-56.32012890625,124.684109375,50],[0.0729625090508734,-0.0775229882995459,0.724063179300088,-0.681468393206874],[0,0,0,0],[8.999999E+09,8.999999E+09,8.999999E+09,8.999999E+09,8.999999E+09,8.999999E+09]];
	LOCAL CONST Robtarget Tr_meulage_bavure_P154 :=[[-53.478453125,125.6220078125,50],[0.118463525450853,-0.126081571718597,0.717791852189305,-0.674421742933433],[0,0,0,0],[8.999999E+09,8.999999E+09,8.999999E+09,8.999999E+09,8.999999E+09,8.999999E+09]];
	LOCAL CONST Robtarget Tr_meulage_bavure_P155 :=[[-53.19229296875,125.72128125,50],[0.161843107852524,-0.172542772115637,0.708656629372146,-0.664711653183692],[0,0,0,0],[8.999999E+09,8.999999E+09,8.999999E+09,8.999999E+09,8.999999E+09,8.999999E+09]];
	LOCAL CONST Robtarget Tr_meulage_bavure_P156 :=[[-53.15704296875,125.74203125,50],[0.201770503470959,-0.215476024990169,0.697411082800909,-0.653051704055641],[0,0,0,0],[8.999999E+09,8.999999E+09,8.999999E+09,8.999999E+09,8.999999E+09,8.999999E+09]];
	LOCAL CONST Robtarget Tr_meulage_bavure_P157 :=[[-51.6136171875,126.909453125,50],[0.23893324300137,-0.255612482203739,0.68436125266746,-0.639705276027888],[0,0,0,0],[8.999999E+09,8.999999E+09,8.999999E+09,8.999999E+09,8.999999E+09,8.999999E+09]];
	LOCAL CONST Robtarget Tr_meulage_bavure_P158 :=[[-50.913359375,127.641875,50],[0.274163476087614,-0.293846352721295,0.669526036119538,-0.62467879452564],[0,0,0,0],[8.999999E+09,8.999999E+09,8.999999E+09,8.999999E+09,8.999999E+09,8.999999E+09]];
	LOCAL CONST Robtarget Tr_meulage_bavure_P159 :=[[-50.3271171875,128.2943125,50],[0.306856273250997,-0.329533851238833,0.653450043134051,-0.608481478421751],[0,0,0,0],[8.999999E+09,8.999999E+09,8.999999E+09,8.999999E+09,8.999999E+09,8.999999E+09]];
	LOCAL CONST Robtarget Tr_meulage_bavure_P160 :=[[-49.6226796875,129.3642265625,50],[0.334370617519238,-0.3598455748161,0.638089189609175,-0.592916215437713],[0,0,0,0],[8.999999E+09,8.999999E+09,8.999999E+09,8.999999E+09,8.999999E+09,8.999999E+09]];
	LOCAL CONST Robtarget Tr_meulage_bavure_P161 :=[[-49.48623828125,129.822359375,50],[0.353015832523773,-0.380805070509742,0.626739583846592,-0.581003282522068],[0,0,0,0],[8.999999E+09,8.999999E+09,8.999999E+09,8.999999E+09,8.999999E+09,8.999999E+09]];
	LOCAL CONST Robtarget Tr_meulage_bavure_P162 :=[[-49.28121875,130.7658046875,50],[0.359659798903472,-0.388984798941856,0.622737188669465,-0.575789934865944],[0,0,0,0],[8.999999E+09,8.999999E+09,8.999999E+09,8.999999E+09,8.999999E+09,8.999999E+09]];
	LOCAL CONST Robtarget Tr_meulage_bavure_P163 :=[[-48.1318671875,137.345796875,50],[0.35233074486465,-0.382167114854553,0.628094602576368,-0.579058298240602],[0,0,0,0],[8.999999E+09,8.999999E+09,8.999999E+09,8.999999E+09,8.999999E+09,8.999999E+09]];
	LOCAL CONST Robtarget Tr_meulage_bavure_P164 :=[[-47.9398203125,138.619296875,50],[0.330224598813358,-0.359352577509282,0.642674753136962,-0.590581578663216],[0,0,0,0],[8.999999E+09,8.999999E+09,8.999999E+09,8.999999E+09,8.999999E+09,8.999999E+09]];
	LOCAL CONST Robtarget Tr_meulage_bavure_P165 :=[[-47.3395078125,140.54565625,50],[0.294093256479054,-0.321197071404187,0.663925882958372,-0.607901324026248],[0,0,0,0],[8.999999E+09,8.999999E+09,8.999999E+09,8.999999E+09,8.999999E+09,8.999999E+09]];
	LOCAL CONST Robtarget Tr_meulage_bavure_P166 :=[[-46.13162109375,142.18496875,50],[0.247189064743329,-0.271060272486718,0.687379117764399,-0.62684435341812],[0,0,0,0],[8.999999E+09,8.999999E+09,8.999999E+09,8.999999E+09,8.999999E+09,8.999999E+09]];
	LOCAL CONST Robtarget Tr_meulage_bavure_P167 :=[[-45.57672265625,143.035765625,50],[0.195256231843547,-0.215065257402255,0.708457141781425,-0.643203247227231],[0,0,0,0],[8.999999E+09,8.999999E+09,8.999999E+09,8.999999E+09,8.999999E+09,8.999999E+09]];
	LOCAL CONST Robtarget Tr_meulage_bavure_P168 :=[[-43.76553515625,143.9645625,50],[0.144336532147658,-0.159754481253507,0.72460351983199,-0.654671834016175],[0,0,0,0],[8.999999E+09,8.999999E+09,8.999999E+09,8.999999E+09,8.999999E+09,8.999999E+09]];
	LOCAL CONST Robtarget Tr_meulage_bavure_P169 :=[[-41.91000390625,144.926109375,50],[0.0983868645310103,-0.109472973240701,0.735662234916882,-0.661163194026025],[0,0,0,0],[8.999999E+09,8.999999E+09,8.999999E+09,8.999999E+09,8.999999E+09,8.999999E+09]];
	LOCAL CONST Robtarget Tr_meulage_bavure_P170 :=[[-40.19134375,145.0563125,50],[0.0588096458830514,-0.0658074126520319,0.742729449315761,-0.66374978351052],[0,0,0,0],[8.999999E+09,8.999999E+09,8.999999E+09,8.999999E+09,8.999999E+09,8.999999E+09]];
	LOCAL CONST Robtarget Tr_meulage_bavure_P171 :=[[-38.67828515625,145.23321875,50],[0.025359252537359,-0.0285473831496346,0.747074705409143,-0.663642478872395],[0,0,0,0],[8.999999E+09,8.999999E+09,8.999999E+09,8.999999E+09,8.999999E+09,8.999999E+09]];
	LOCAL CONST Robtarget Tr_meulage_bavure_P172 :=[[-38.5074765625,145.219359375,50],[0.00260949525945307,-0.00295606697395452,-0.74968091670879,0.661787711675885],[0,0,0,0],[8.999999E+09,8.999999E+09,8.999999E+09,8.999999E+09,8.999999E+09,8.999999E+09]];
	LOCAL CONST Robtarget Tr_meulage_bavure_P173 :=[[-35.6859453125,144.576109375,50],[0.0255699285650557,-0.0291553658002909,-0.751256905903433,0.658869641682351],[0,0,0,0],[8.999999E+09,8.999999E+09,8.999999E+09,8.999999E+09,8.999999E+09,8.999999E+09]];
	LOCAL CONST Robtarget Tr_meulage_bavure_P174 :=[[-33.7073984375,144.214296875,50],[0.0437880503605696,-0.050262484630657,-0.752322367423892,0.655413872875821],[0,0,0,0],[8.999999E+09,8.999999E+09,8.999999E+09,8.999999E+09,8.999999E+09,8.999999E+09]];
	LOCAL CONST Robtarget Tr_meulage_bavure_P175 :=[[-33.01946875,144.0430625,50],[0.0575367856107434,-0.066490959455461,-0.753259279022407,0.651819706037582],[0,0,0,0],[8.999999E+09,8.999999E+09,8.999999E+09,8.999999E+09,8.999999E+09,8.999999E+09]];
	LOCAL CONST Robtarget Tr_meulage_bavure_P176 :=[[-27.1693125,142.589390625,50],[0.0673409158431606,-0.0783473834870864,-0.754308291311531,0.648340875013145],[0,0,0,0],[8.999999E+09,8.999999E+09,8.999999E+09,8.999999E+09,8.999999E+09,8.999999E+09]];
	LOCAL CONST Robtarget Tr_meulage_bavure_P177 :=[[-25.4131171875,142.19815625,50],[0.0739384542429228,-0.0865981765125488,-0.755560827094071,0.645105958250109],[0,0,0,0],[8.999999E+09,8.999999E+09,8.999999E+09,8.999999E+09,8.999999E+09,8.999999E+09]];
	LOCAL CONST Robtarget Tr_meulage_bavure_P178 :=[[-19.949828125,140.875390625,50],[0.0782294206585914,-0.0922208328134283,-0.756988079908947,0.642140578545216],[0,0,0,0],[8.999999E+09,8.999999E+09,8.999999E+09,8.999999E+09,8.999999E+09,8.999999E+09]];
	LOCAL CONST Robtarget Tr_meulage_bavure_P179 :=[[-19.50540234375,140.785640625,50],[0.0810714654472885,-0.0961706723788441,-0.758503212555855,0.639414963702663],[0,0,0,0],[8.999999E+09,8.999999E+09,8.999999E+09,8.999999E+09,8.999999E+09,8.999999E+09]];
	LOCAL CONST Robtarget Tr_meulage_bavure_P180 :=[[-16.86636328125,140.10646875,50],[0.0830839175144657,-0.0991457171555351,-0.76002046190916,0.636895664060881],[0,0,0,0],[8.999999E+09,8.999999E+09,8.999999E+09,8.999999E+09,8.999999E+09,8.999999E+09]];
	LOCAL CONST Robtarget Tr_meulage_bavure_P181 :=[[-9.1235048828125,137.943109375,50],[0.0846191865819513,-0.101544143504816,-0.761484113426329,0.634563097872386],[0,0,0,0],[8.999999E+09,8.999999E+09,8.999999E+09,8.999999E+09,8.999999E+09,8.999999E+09]];
	LOCAL CONST Robtarget Tr_meulage_bavure_P182 :=[[-6.4043271484375,137.1874375,50],[0.0858024688595693,-0.103498573502936,-0.762862698865075,0.632429034991875],[0,0,0,0],[8.999999E+09,8.999999E+09,8.999999E+09,8.999999E+09,8.999999E+09,8.999999E+09]];
	LOCAL CONST Robtarget Tr_meulage_bavure_P183 :=[[-3.73745727539063,136.470890625,50],[0.0866431535850849,-0.105007531361487,-0.764149023872507,0.630509834664688],[0,0,0,0],[8.999999E+09,8.999999E+09,8.999999E+09,8.999999E+09,8.999999E+09,8.999999E+09]];
	LOCAL CONST Robtarget Tr_meulage_bavure_P184 :=[[-2.75320434570313,136.16375,50],[0.0871015461292202,-0.10601407794586,-0.765352452508939,0.628816316087409],[0,0,0,0],[8.999999E+09,8.999999E+09,8.999999E+09,8.999999E+09,8.999999E+09,8.999999E+09]];
	LOCAL CONST Robtarget Tr_meulage_bavure_P185 :=[[-0.1947021484375,135.414,50],[0.087184523297091,-0.106516079515365,-0.766466762769312,0.627361048577345],[0,0,0,0],[8.999999E+09,8.999999E+09,8.999999E+09,8.999999E+09,8.999999E+09,8.999999E+09]];
	LOCAL CONST Robtarget Tr_meulage_bavure_P186 :=[[4.61236572265625,134.06759375,50],[0.0869586966798894,-0.106587987257267,-0.767479864047654,0.626140434986892],[0,0,0,0],[8.999999E+09,8.999999E+09,8.999999E+09,8.999999E+09,8.999999E+09,8.999999E+09]];
	LOCAL CONST Robtarget Tr_meulage_bavure_P187 :=[[11.3466796875,132.23821875,50],[0.0865249361086305,-0.10635250383225,-0.768383342248204,0.625131681900292],[0,0,0,0],[8.999999E+09,8.999999E+09,8.999999E+09,8.999999E+09,8.999999E+09,8.999999E+09]];
	LOCAL CONST Robtarget Tr_meulage_bavure_P188 :=[[20.052947265625,129.9318828125,50],[0.0860014136700688,-0.105951822717768,-0.769153554340039,0.624324257061679],[0,0,0,0],[8.999999E+09,8.999999E+09,8.999999E+09,8.999999E+09,8.999999E+09,8.999999E+09]];
	LOCAL CONST Robtarget Tr_meulage_bavure_P189 :=[[26.43633984375,128.110078125,50],[0.0854868584931577,-0.105508652420373,-0.76977729905776,0.62370091481795],[0,0,0,0],[8.999999E+09,8.999999E+09,8.999999E+09,8.999999E+09,8.999999E+09,8.999999E+09]];
	LOCAL CONST Robtarget Tr_meulage_bavure_P190 :=[[29.66665625,127.2478359375,50],[0.0850579054559104,-0.105121174586693,-0.770249992142775,0.623241238187127],[0,0,0,0],[8.999999E+09,8.999999E+09,8.999999E+09,8.999999E+09,8.999999E+09,8.999999E+09]];
	LOCAL CONST Robtarget Tr_meulage_bavure_P191 :=[[33.7070625,126.195828125,50],[0.0847805841323715,-0.104873944720326,-0.770566408740507,0.622929464701847],[0,0,0,0],[8.999999E+09,8.999999E+09,8.999999E+09,8.999999E+09,8.999999E+09,8.999999E+09]];
	LOCAL CONST Robtarget Tr_meulage_bavure_P192 :=[[40.50408984375,124.2788125,50],[0.0847105054444159,-0.104837397083956,-0.770719740827311,0.622755434772829],[0,0,0,0],[8.999999E+09,8.999999E+09,8.999999E+09,8.999999E+09,8.999999E+09,8.999999E+09]];
	LOCAL CONST Robtarget Tr_meulage_bavure_P193 :=[[41.45681640625,123.9972265625,50],[0.0848859800573526,-0.105060984513183,-0.770708244620949,0.622708086984679],[0,0,0,0],[8.999999E+09,8.999999E+09,8.999999E+09,8.999999E+09,8.999999E+09,8.999999E+09]];
	LOCAL CONST Robtarget Tr_meulage_bavure_P194 :=[[48.29797265625,122.1701640625,50],[0.0853054944357664,-0.105546436381405,-0.770542703581653,0.622773525724507],[0,0,0,0],[8.999999E+09,8.999999E+09,8.999999E+09,8.999999E+09,8.999999E+09,8.999999E+09]];
	LOCAL CONST Robtarget Tr_meulage_bavure_P195 :=[[51.30578515625,121.4099765625,50],[0.0859140025543379,-0.106225385664739,-0.770233475769126,0.622956936240445],[0,0,0,0],[8.999999E+09,8.999999E+09,8.999999E+09,8.999999E+09,8.999999E+09,8.999999E+09]];
	LOCAL CONST Robtarget Tr_meulage_bavure_P196 :=[[54.328828125,120.690671875,50],[0.0866207249454984,-0.106986565363642,-0.769801363197173,0.623262854710099],[0,0,0,0],[8.999999E+09,8.999999E+09,8.999999E+09,8.999999E+09,8.999999E+09,8.999999E+09]];
	LOCAL CONST Robtarget Tr_meulage_bavure_P197 :=[[62.490296875,118.2496953125,50],[0.0873315948856018,-0.107716099250654,-0.769271361661927,0.623692237103979],[0,0,0,0],[8.999999E+09,8.999999E+09,8.999999E+09,8.999999E+09,8.999999E+09,8.999999E+09]];
	LOCAL CONST Robtarget Tr_meulage_bavure_P198 :=[[64.112,117.80203125,50],[0.0880026317724586,-0.108361854951403,-0.768658444540542,0.624241492396273],[0,0,0,0],[8.999999E+09,8.999999E+09,8.999999E+09,8.999999E+09,8.999999E+09,8.999999E+09]];
	LOCAL CONST Robtarget Tr_meulage_bavure_P199 :=[[66.6199609375,117.068453125,50],[0.0886595335972033,-0.108954197032184,-0.767955580925725,0.62491015016275],[0,0,0,0],[8.999999E+09,8.999999E+09,8.999999E+09,8.999999E+09,8.999999E+09,8.999999E+09]];
	LOCAL CONST Robtarget Tr_meulage_bavure_P200 :=[[68.724515625,116.4675,50],[0.0893689800751286,-0.109578831263464,-0.76716269569306,0.625673288127455],[0,0,0,0],[8.999999E+09,8.999999E+09,8.999999E+09,8.999999E+09,8.999999E+09,8.999999E+09]];
	LOCAL CONST Robtarget Tr_meulage_bavure_P201 :=[[69.4386328125,116.3375859375,50],[0.0902010944837394,-0.110325746305937,-0.766280886330359,0.626502669986915],[0,0,0,0],[8.999999E+09,8.999999E+09,8.999999E+09,8.999999E+09,8.999999E+09,8.999999E+09]];
	LOCAL CONST Robtarget Tr_meulage_bavure_P202 :=[[71.799984375,115.6488671875,50],[0.0911693830467795,-0.111211051035518,-0.765310416759655,0.627391593601323],[0,0,0,0],[8.999999E+09,8.999999E+09,8.999999E+09,8.999999E+09,8.999999E+09,8.999999E+09]];
	LOCAL CONST Robtarget Tr_meulage_bavure_P203 :=[[77.7030625,113.9541328125,50],[0.0921982996625046,-0.112142573276133,-0.764268262078093,0.628345080651135],[0,0,0,0],[8.999999E+09,8.999999E+09,8.999999E+09,8.999999E+09,8.999999E+09,8.999999E+09]];
	LOCAL CONST Robtarget Tr_meulage_bavure_P204 :=[[85.047671875,111.8714296875,50],[0.0931310126895317,-0.1129332017187,-0.763193266717335,0.629371705800562],[0,0,0,0],[8.999999E+09,8.999999E+09,8.999999E+09,8.999999E+09,8.999999E+09,8.999999E+09]];
	LOCAL CONST Robtarget Tr_meulage_bavure_P205 :=[[85.66396875,111.708953125,50],[0.0937768885143333,-0.113356646990108,-0.762128820121454,0.630488562389526],[0,0,0,0],[8.999999E+09,8.999999E+09,8.999999E+09,8.999999E+09,8.999999E+09,8.999999E+09]];
	LOCAL CONST Robtarget Tr_meulage_bavure_P206 :=[[86.0647578125,111.5926796875,50],[0.0939803414534468,-0.113232244257156,-0.761112522002446,0.631707118158294],[0,0,0,0],[8.999999E+09,8.999999E+09,8.999999E+09,8.999999E+09,8.999999E+09,8.999999E+09]];
	LOCAL CONST Robtarget Tr_meulage_bavure_P207 :=[[94.03115625,109.136171875,50],[0.0936866526623541,-0.11249948118263,-0.76015295009662,0.633035678541082],[0,0,0,0],[8.999999E+09,8.999999E+09,8.999999E+09,8.999999E+09,8.999999E+09,8.999999E+09]];
	LOCAL CONST Robtarget Tr_meulage_bavure_P208 :=[[96.7705390625,108.3211953125,50],[0.0930028021900812,-0.111294009407425,-0.759232616658954,0.634452485262695],[0,0,0,0],[8.999999E+09,8.999999E+09,8.999999E+09,8.999999E+09,8.999999E+09,8.999999E+09]];
	LOCAL CONST Robtarget Tr_meulage_bavure_P209 :=[[99.577453125,107.4735703125,50],[0.0922063530079866,-0.109953724137246,-0.75830566513492,0.635909337278203],[0,0,0,0],[8.999999E+09,8.999999E+09,8.999999E+09,8.999999E+09,8.999999E+09,8.999999E+09]];
	LOCAL CONST Robtarget Tr_meulage_bavure_P210 :=[[103.5093671875,106.3269375,50],[0.0917213060005248,-0.108982846344829,-0.757295282252709,0.637349038365892],[0,0,0,0],[8.999999E+09,8.999999E+09,8.999999E+09,8.999999E+09,8.999999E+09,8.999999E+09]];
	LOCAL CONST Robtarget Tr_meulage_bavure_P211 :=[[109.3239765625,104.6611953125,50],[0.0920122482902498,-0.108925820207777,-0.756119068393039,0.638711880482178],[0,0,0,0],[8.999999E+09,8.999999E+09,8.999999E+09,8.999999E+09,8.999999E+09,8.999999E+09]];
	LOCAL CONST Robtarget Tr_meulage_bavure_P212 :=[[112.0927109375,103.9254765625,50],[0.0934364831575626,-0.110189957979828,-0.754705578509744,0.639958816285723],[0,0,0,0],[8.999999E+09,8.999999E+09,8.999999E+09,8.999999E+09,8.999999E+09,8.999999E+09]];
	LOCAL CONST Robtarget Tr_meulage_bavure_P213 :=[[116.5132421875,102.7547578125,50],[0.0960542151858976,-0.112830352282311,-0.753038880396986,0.641073587008017],[0,0,0,0],[8.999999E+09,8.999999E+09,8.999999E+09,8.999999E+09,8.999999E+09,8.999999E+09]];
	LOCAL CONST Robtarget Tr_meulage_bavure_P214 :=[[119.901125,101.886234375,50],[0.0994585543511626,-0.116348629856775,-0.751166542236914,0.642121342209296],[0,0,0,0],[8.999999E+09,8.999999E+09,8.999999E+09,8.999999E+09,8.999999E+09,8.999999E+09]];
	LOCAL CONST Robtarget Tr_meulage_bavure_P215 :=[[123.742734375,100.759859375,50],[0.102797737234972,-0.119732773666272,-0.749218219911941,0.643248588868668],[0,0,0,0],[8.999999E+09,8.999999E+09,8.999999E+09,8.999999E+09,8.999999E+09,8.999999E+09]];
	LOCAL CONST Robtarget Tr_meulage_bavure_P216 :=[[128.8837890625,99.2673984375,50],[0.104980171945493,-0.1217147031486,-0.747398869782906,0.64463914245334],[0,0,0,0],[8.999999E+09,8.999999E+09,8.999999E+09,8.999999E+09,8.999999E+09,8.999999E+09]];
	LOCAL CONST Robtarget Tr_meulage_bavure_P217 :=[[129.5076875,98.9887421875,50],[0.105028512903552,-0.121181030141381,-0.745894122526642,0.646472062344038],[0,0,0,0],[8.999999E+09,8.999999E+09,8.999999E+09,8.999999E+09,8.999999E+09,8.999999E+09]];
	LOCAL CONST Robtarget Tr_meulage_bavure_P218 :=[[131.35796875,98.4144609375,50],[0.10249779346123,-0.117652269531182,-0.744761923808864,0.648831120288062],[0,0,0,0],[8.999999E+09,8.999999E+09,8.999999E+09,8.999999E+09,8.999999E+09,8.999999E+09]];
	LOCAL CONST Robtarget Tr_meulage_bavure_P219 :=[[134.117125,97.6161796875,50],[0.0977400920483205,-0.11157998876392,-0.743895463797094,0.65162590453107],[0,0,0,0],[8.999999E+09,8.999999E+09,8.999999E+09,8.999999E+09,8.999999E+09,8.999999E+09]];
	LOCAL CONST Robtarget Tr_meulage_bavure_P220 :=[[135.51721875,97.226046875,50],[0.0918613941703946,-0.104266963915484,-0.743053595302287,0.654645888252011],[0,0,0,0],[8.999999E+09,8.999999E+09,8.999999E+09,8.999999E+09,8.999999E+09,8.999999E+09]];
	LOCAL CONST Robtarget Tr_meulage_bavure_P221 :=[[138.0495625,96.6037890625,50],[0.0863786360676273,-0.0974527086049605,-0.741974087712015,0.657659603427622],[0,0,0,0],[8.999999E+09,8.999999E+09,8.999999E+09,8.999999E+09,8.999999E+09,8.999999E+09]];
	LOCAL CONST Robtarget Tr_meulage_bavure_P222 :=[[142.0440625,95.5323828125,50],[0.0826508913482682,-0.092660011157343,-0.740487784880716,0.660500411002225],[0,0,0,0],[8.999999E+09,8.999999E+09,8.999999E+09,8.999999E+09,8.999999E+09,8.999999E+09]];
	LOCAL CONST Robtarget Tr_meulage_bavure_P223 :=[[142.262078125,95.513734375,50],[0.0814296925342413,-0.0906972875290771,-0.738552630495336,0.663086132562782],[0,0,0,0],[8.999999E+09,8.999999E+09,8.999999E+09,8.999999E+09,8.999999E+09,8.999999E+09]];
	LOCAL CONST Robtarget Tr_meulage_bavure_P224 :=[[151.236640625,92.7137734375,50],[0.0826296344217782,-0.0914242360742305,-0.736234323716048,0.665411882337504],[0,0,0,0],[8.999999E+09,8.999999E+09,8.999999E+09,8.999999E+09,8.999999E+09,8.999999E+09]];
	LOCAL CONST Robtarget Tr_meulage_bavure_P225 :=[[152.364875,92.365265625,50],[0.0855609137014986,-0.0940340464717138,-0.733642924081411,0.667536506938758],[0,0,0,0],[8.999999E+09,8.999999E+09,8.999999E+09,8.999999E+09,8.999999E+09,8.999999E+09]];
	LOCAL CONST Robtarget Tr_meulage_bavure_P226 :=[[152.630609375,92.2931796875,50],[0.0895621778242674,-0.0977739110488583,-0.730883321128435,0.669498655351789],[0,0,0,0],[8.999999E+09,8.999999E+09,8.999999E+09,8.999999E+09,8.999999E+09,8.999999E+09]];
	LOCAL CONST Robtarget Tr_meulage_bavure_P227 :=[[153.1405,92.136625,50],[0.0944579436771033,-0.102444689518096,-0.728011239397273,0.671254361458517],[0,0,0,0],[8.999999E+09,8.999999E+09,8.999999E+09,8.999999E+09,8.999999E+09,8.999999E+09]];
	LOCAL CONST Robtarget Tr_meulage_bavure_P228 :=[[155.846625,91.4085078125,50],[0.100989710670536,-0.108837899588145,-0.724917299300571,0.672644258971032],[0,0,0,0],[8.999999E+09,8.999999E+09,8.999999E+09,8.999999E+09,8.999999E+09,8.999999E+09]];
	LOCAL CONST Robtarget Tr_meulage_bavure_P229 :=[[159.151734375,90.6287265625,50],[0.110819668117851,-0.118716494301188,-0.721296839145693,0.673317358292148],[0,0,0,0],[8.999999E+09,8.999999E+09,8.999999E+09,8.999999E+09,8.999999E+09,8.999999E+09]];
	LOCAL CONST Robtarget Tr_meulage_bavure_P230 :=[[160.38396875,90.3316640625,50],[0.126122814859885,-0.134357583547145,-0.716610250020207,0.672689248376372],[0,0,0,0],[8.999999E+09,8.999999E+09,8.999999E+09,8.999999E+09,8.999999E+09,8.999999E+09]];
	LOCAL CONST Robtarget Tr_meulage_bavure_P231 :=[[161.1148125,90.0939609375,50],[0.148950748649148,-0.157871810936768,-0.710019416452882,0.669897450396934],[0,0,0,0],[8.999999E+09,8.999999E+09,8.999999E+09,8.999999E+09,8.999999E+09,8.999999E+09]];
	LOCAL CONST Robtarget Tr_meulage_bavure_P232 :=[[162.89178125,89.49334375,50],[0.180238998057261,-0.19017038386354,-0.700448343542026,0.663868395625022],[0,0,0,0],[8.999999E+09,8.999999E+09,8.999999E+09,8.999999E+09,8.999999E+09,8.999999E+09]];
	LOCAL CONST Robtarget Tr_meulage_bavure_P233 :=[[163.99846875,89.1625078125,50],[0.219056817826717,-0.230223102146587,-0.686902988719632,0.653586809758025],[0,0,0,0],[8.999999E+09,8.999999E+09,8.999999E+09,8.999999E+09,8.999999E+09,8.999999E+09]];
	LOCAL CONST Robtarget Tr_meulage_bavure_P234 :=[[166.530515625,87.3825078125,50],[0.262472383800806,-0.274945563373132,-0.66903056732987,0.638679328694476],[0,0,0,0],[8.999999E+09,8.999999E+09,8.999999E+09,8.999999E+09,8.999999E+09,8.999999E+09]];
	LOCAL CONST Robtarget Tr_meulage_bavure_P235 :=[[166.927375,87.1272265625,50],[0.306650629514095,-0.320368475913498,-0.647480848557644,0.619756389084086],[0,0,0,0],[8.999999E+09,8.999999E+09,8.999999E+09,8.999999E+09,8.999999E+09,8.999999E+09]];
	LOCAL CONST Robtarget Tr_meulage_bavure_P236 :=[[167.023625,86.9859296875,50],[0.34864753653045,-0.363494936342623,-0.623467152578671,0.598000866370581],[0,0,0,0],[8.999999E+09,8.999999E+09,8.999999E+09,8.999999E+09,8.999999E+09,8.999999E+09]];
	LOCAL CONST Robtarget Tr_meulage_bavure_P237 :=[[168.406375,84.2996796875,50],[0.387119559668182,-0.403007112239651,-0.598067506937531,0.574490183686455],[0,0,0,0],[8.999999E+09,8.999999E+09,8.999999E+09,8.999999E+09,8.999999E+09,8.999999E+09]];
	LOCAL CONST Robtarget Tr_meulage_bavure_P238 :=[[168.427921875,84.1041875,50],[0.421760562527715,-0.438646089352045,-0.572020197675838,0.550000481493752],[0,0,0,0],[8.999999E+09,8.999999E+09,8.999999E+09,8.999999E+09,8.999999E+09,8.999999E+09]];
	LOCAL CONST Robtarget Tr_meulage_bavure_P239 :=[[168.736640625,82.6158125,50],[0.452430882393441,-0.470300659600423,-0.546055125840183,0.525306944347551],[0,0,0,0],[8.999999E+09,8.999999E+09,8.999999E+09,8.999999E+09,8.999999E+09,8.999999E+09]];
	LOCAL CONST Robtarget Tr_meulage_bavure_P240 :=[[168.560125,80.3153984375,50],[0.478743526266297,-0.49757700373529,-0.521248703078886,0.501519242851659],[0,0,0,0],[8.999999E+09,8.999999E+09,8.999999E+09,8.999999E+09,8.999999E+09,8.999999E+09]];
	LOCAL CONST Robtarget Tr_meulage_bavure_P241 :=[[168.562015625,79.8987109375,50],[0.500317378564995,-0.52007342017413,-0.498876370336502,0.479925541572974],[0,0,0,0],[8.999999E+09,8.999999E+09,8.999999E+09,8.999999E+09,8.999999E+09,8.999999E+09]];
	LOCAL CONST Robtarget Tr_meulage_bavure_P242 :=[[168.383734375,78.884828125,50],[0.517070628377123,-0.537684082378158,-0.480033049672985,0.46162979111892],[0,0,0,0],[8.999999E+09,8.999999E+09,8.999999E+09,8.999999E+09,8.999999E+09,8.999999E+09]];
	LOCAL CONST Robtarget Tr_meulage_bavure_P243 :=[[168.15515625,78.1168828125,50],[0.529321040531053,-0.550702393890604,-0.465313052939919,0.447246992363294],[0,0,0,0],[8.999999E+09,8.999999E+09,8.999999E+09,8.999999E+09,8.999999E+09,8.999999E+09]];
	LOCAL CONST Robtarget Tr_meulage_bavure_P244 :=[[167.710515625,76.159453125,50],[0.537709913069671,-0.559752388298682,-0.454702226172844,0.43679651863767],[0,0,0,0],[8.999999E+09,8.999999E+09,8.999999E+09,8.999999E+09,8.999999E+09,8.999999E+09]];
	LOCAL CONST Robtarget Tr_meulage_bavure_P245 :=[[167.502203125,75.067046875,50],[0.542978981138286,-0.565574965878791,-0.447772029071907,0.429882535111699],[0,0,0,0],[8.999999E+09,8.999999E+09,8.999999E+09,8.999999E+09,8.999999E+09,8.999999E+09]];
	LOCAL CONST Robtarget Tr_meulage_bavure_P246 :=[[167.066953125,73.6228359375,50],[0.545906854289828,-0.568971564598597,-0.443791170167035,0.425800965709782],[0,0,0,0],[8.999999E+09,8.999999E+09,8.999999E+09,8.999999E+09,8.999999E+09,8.999999E+09]];
	LOCAL CONST Robtarget Tr_meulage_bavure_P247 :=[[166.529484375,71.6883828125,50],[0.547261304635725,-0.570708426352787,-0.441877380616225,0.423723184447198],[0,0,0,0],[8.999999E+09,8.999999E+09,8.999999E+09,8.999999E+09,8.999999E+09,8.999999E+09]];
	LOCAL CONST Robtarget Tr_meulage_bavure_P248 :=[[165.0523125,66.31634375,50],[0.547717055481567,-0.5714763087711,-0.441173632434147,0.422831741586202],[0,0,0,0],[8.999999E+09,8.999999E+09,8.999999E+09,8.999999E+09,8.999999E+09,8.999999E+09]];
	LOCAL CONST Robtarget Tr_meulage_bavure_P249 :=[[164.558953125,64.43182421875,50],[0.547816145163016,-0.57184777947627,-0.440957470653158,0.422426440083905],[0,0,0,0],[8.999999E+09,8.999999E+09,8.999999E+09,8.999999E+09,8.999999E+09,8.999999E+09]];
	LOCAL CONST Robtarget Tr_meulage_bavure_P250 :=[[164.444390625,63.9650859375,50],[0.547863453398091,-0.572153932702597,-0.440814328921402,0.422099799977735],[0,0,0,0],[8.999999E+09,8.999999E+09,8.999999E+09,8.999999E+09,8.999999E+09,8.999999E+09]];
	LOCAL CONST Robtarget Tr_meulage_bavure_P251 :=[[164.072203125,62.642546875,50],[0.547963387599864,-0.572505452985805,-0.440602306459617,0.421714642494264],[0,0,0,0],[8.999999E+09,8.999999E+09,8.999999E+09,8.999999E+09,8.999999E+09,8.999999E+09]];
	LOCAL CONST Robtarget Tr_meulage_bavure_P252 :=[[163.193234375,59.6897578125,50],[0.548067490613862,-0.572859454886323,-0.440384614033586,0.421325838754353],[0,0,0,0],[8.999999E+09,8.999999E+09,8.999999E+09,8.999999E+09,8.999999E+09,8.999999E+09]];
	LOCAL CONST Robtarget Tr_meulage_bavure_P253 :=[[162.273921875,56.48968359375,50],[0.548054492116352,-0.573105877434887,-0.440321089686516,0.421073942316495],[0,0,0,0],[8.999999E+09,8.999999E+09,8.999999E+09,8.999999E+09,8.999999E+09,8.999999E+09]];
	LOCAL CONST Robtarget Tr_meulage_bavure_P254 :=[[161.7705625,54.75924609375,50],[0.547857822210366,-0.573184575896671,-0.440499787548265,0.421035848553305],[0,0,0,0],[8.999999E+09,8.999999E+09,8.999999E+09,8.999999E+09,8.999999E+09,8.999999E+09]];
	LOCAL CONST Robtarget Tr_meulage_bavure_P255 :=[[158.91828125,44.34161328125,50],[0.547506357516806,-0.573128599339125,-0.440880598093385,0.421170624952727],[0,0,0,0],[8.999999E+09,8.999999E+09,8.999999E+09,8.999999E+09,8.999999E+09,8.999999E+09]];
	LOCAL CONST Robtarget Tr_meulage_bavure_P256 :=[[156.758671875,36.10925390625,50],[0.547102471132479,-0.573055978639264,-0.441320643910947,0.421333384251185],[0,0,0,0],[8.999999E+09,8.999999E+09,8.999999E+09,8.999999E+09,8.999999E+09,8.999999E+09]];
	LOCAL CONST Robtarget Tr_meulage_bavure_P257 :=[[156.16296875,33.7295546875,50],[0.546778962526323,-0.573106266107689,-0.441639165346887,0.421351185495479],[0,0,0,0],[8.999999E+09,8.999999E+09,8.999999E+09,8.999999E+09,8.999999E+09,8.999999E+09]];
	LOCAL CONST Robtarget Tr_meulage_bavure_P258 :=[[155.43646875,30.9241953125,50],[0.546645197679891,-0.573376972546252,-0.441692702018425,0.421100263821896],[0,0,0,0],[8.999999E+09,8.999999E+09,8.999999E+09,8.999999E+09,8.999999E+09,8.999999E+09]];
	LOCAL CONST Robtarget Tr_meulage_bavure_P259 :=[[153.489984375,23.12323046875,50],[0.546734089123416,-0.573904631079155,-0.44143495060465,0.420535961126938],[0,0,0,0],[8.999999E+09,8.999999E+09,8.999999E+09,8.999999E+09,8.999999E+09,8.999999E+09]];
	LOCAL CONST Robtarget Tr_meulage_bavure_P260 :=[[150.613640625,12.741515625,50],[0.547012135300881,-0.574648440956601,-0.440911513903558,0.419706957348805],[0,0,0,0],[8.999999E+09,8.999999E+09,8.999999E+09,8.999999E+09,8.999999E+09,8.999999E+09]];
	LOCAL CONST Robtarget Tr_meulage_bavure_P261 :=[[150.054328125,10.692931640625,50],[0.547409409977123,-0.575511832127871,-0.440223398456239,0.418727152691295],[0,0,0,0],[8.999999E+09,8.999999E+09,8.999999E+09,8.999999E+09,8.999999E+09,8.999999E+09]];
	LOCAL CONST Robtarget Tr_meulage_bavure_P262 :=[[149.692625,9.3722841796875,50],[0.547828312980544,-0.576377511474761,-0.439508350272666,0.417738571122721],[0,0,0,0],[8.999999E+09,8.999999E+09,8.999999E+09,8.999999E+09,8.999999E+09,8.999999E+09]];
	LOCAL CONST Robtarget Tr_meulage_bavure_P263 :=[[148.613703125,5.2665712890625,50],[0.548175483882057,-0.577134548002692,-0.438899738558927,0.416876926520653],[0,0,0,0],[8.999999E+09,8.999999E+09,8.999999E+09,8.999999E+09,8.999999E+09,8.999999E+09]];
	LOCAL CONST Robtarget Tr_meulage_bavure_P264 :=[[146.364203125,-3.26248168945313,50],[0.548380445988877,-0.577695207381415,-0.438501187985519,0.416249735088052],[0,0,0,0],[8.999999E+09,8.999999E+09,8.999999E+09,8.999999E+09,8.999999E+09,8.999999E+09]];
	LOCAL CONST Robtarget Tr_meulage_bavure_P265 :=[[144.30578125,-10.2499697265625,50],[0.548406939297358,-0.578006817968467,-0.438369667680023,0.415920643597524],[0,0,0,0],[8.999999E+09,8.999999E+09,8.999999E+09,8.999999E+09,8.999999E+09,8.999999E+09]];
	LOCAL CONST Robtarget Tr_meulage_bavure_P266 :=[[142.754828125,-15.587982421875,50],[0.548253313533703,-0.578056978434944,-0.438512190644615,0.415903224967105],[0,0,0,0],[8.999999E+09,8.999999E+09,8.999999E+09,8.999999E+09,8.999999E+09,8.999999E+09]];
	LOCAL CONST Robtarget Tr_meulage_bavure_P267 :=[[141.558953125,-20.13653515625,50],[0.547940072223752,-0.577866738186702,-0.438900534570051,0.416170675207918],[0,0,0,0],[8.999999E+09,8.999999E+09,8.999999E+09,8.999999E+09,8.999999E+09,8.999999E+09]];
	LOCAL CONST Robtarget Tr_meulage_bavure_P268 :=[[139.748109375,-27.11804296875,50],[0.547508730983152,-0.577476936799646,-0.439477237126479,0.416670535326645],[0,0,0,0],[8.999999E+09,8.999999E+09,8.999999E+09,8.999999E+09,8.999999E+09,8.999999E+09]];
